# B&R Automation Studio project VisionSample (part 8)

#### ViSaveImgOnPlc.st
```iecst
// Note: This FBK needs to be called at least once in the INIT of the task to alloc memory (restriction of AsMem)
FUNCTION_BLOCK ViSaveImgOnPlc
	IF MemInfo.SvgAdr = 0 THEN // This will only be done once in the INIT of the task
		// Create memory for uploading and transforming image
		// Size: a 5MP picture in bmp format has less than 6.000.000 Bytes. A SVG with bas64 conversion maximum the 4/3 size.
		MemInfo.UploadSize			:= 6000000;		// Upload of the picture data with httpClient
		MemInfo.SvgHeaderSize		:= 2000; 		// Fileheader, ...
		MemInfo.CrosshSize			:= 18000; 		// Crosshairs, Texts, ...
		MemInfo.SvgSize				:= MemInfo.UploadSize * 4 / 3 + MemInfo.SvgHeaderSize + MemInfo.CrosshSize;
		AsMemPartCreate_0.enable	:= TRUE;
		AsMemPartCreate_0.len		:= MemInfo.UploadSize + MemInfo.SvgSize + MemInfo.CrosshSize + 1000; // 1000 Bytes for AsMemPart stuff/header
		AsMemPartCreate_0();
		IF AsMemPartCreate_0.status = ERR_OK THEN
			// Upload mem for loading the image from camera to plc
			AsMemPartAllocClear_0.len		:= MemInfo.UploadSize;
			AsMemPartAllocClear_0(enable := TRUE, ident := AsMemPartCreate_0.ident);
			IF AsMemPartAllocClear_0.status = ERR_OK THEN
				MemInfo.UploadAdr			:= AsMemPartAllocClear_0.mem;
			END_IF
			// Svg mem for creating the svg file including the image
			AsMemPartAllocClear_0.len		:= MemInfo.SvgSize;
			AsMemPartAllocClear_0(enable := TRUE, ident := AsMemPartCreate_0.ident);
			IF AsMemPartAllocClear_0.status = ERR_OK THEN
				MemInfo.SvgAdr 				:= AsMemPartAllocClear_0.mem;
			END_IF
			// Mem for creating the crosshaurs
			AsMemPartAllocClear_0.len		:= MemInfo.CrosshSize;
			AsMemPartAllocClear_0(enable := TRUE, ident := AsMemPartCreate_0.ident);
			IF AsMemPartAllocClear_0.status = ERR_OK THEN
				MemInfo.CrosshAdr			:= AsMemPartAllocClear_0.mem;
			END_IF
		END_IF
	END_IF
	IF NOT Enable THEN
		Status := ERR_FUB_ENABLE_FALSE;
		Step := 0;
		RETURN;
	END_IF
	CASE Step OF
		0:
			Status := ERR_FUB_BUSY;
			IF MemInfo.UploadAdr <> 0 AND MemInfo.SvgAdr <> 0 AND MemInfo.CrosshAdr <> 0 THEN
				Step := 1;
			END_IF
		1: // Initialization
			ACTION_InitTexts;
			brsmemcpy(ADR(b64key), ADR('ABCDEFGHIJKLMNOPQRSTUVWXYZabcdefghijklmnopqrstuvwxyz0123456789+/'), SIZEOF(b64key));
			// Generate new filenames
			DTGetTime_0(enable := TRUE);
			DT_TO_DTStructure(DTGetTime_0.DT1, ADR(DTStructure_0));
			FileNameImg := CFG.DirName;
			brsstrcat(ADR(FileNameImg), ADR('/'));
			tmpStr1 := UINT_TO_STRING(DTStructure_0.year);
			brsstrcat(ADR(FileNameImg), ADR(tmpStr1));
			brsstrcat(ADR(FileNameImg), ADR('_'));
			tmpStr1 := USINT_TO_STRING(DTStructure_0.month);
			IF(DTStructure_0.month < 10) THEN
				brsstrcat(ADR(FileNameImg), ADR('0'));
			END_IF
			brsstrcat(ADR(FileNameImg), ADR(tmpStr1));
			brsstrcat(ADR(FileNameImg), ADR('_'));
			tmpStr1 := USINT_TO_STRING(DTStructure_0.day);
			IF(DTStructure_0.day < 10) THEN
				brsstrcat(ADR(FileNameImg), ADR('0'));
			END_IF
			brsstrcat(ADR(FileNameImg), ADR(tmpStr1));
			brsstrcat(ADR(FileNameImg), ADR('_'));
			tmpStr1 := USINT_TO_STRING(DTStructure_0.hour);
			IF(DTStructure_0.hour < 10) THEN
				brsstrcat(ADR(FileNameImg), ADR('0'));
			END_IF
			brsstrcat(ADR(FileNameImg), ADR(tmpStr1));
			brsstrcat(ADR(FileNameImg), ADR('_'));
			tmpStr1 := USINT_TO_STRING(DTStructure_0.minute);
			IF(DTStructure_0.minute < 10) THEN
				brsstrcat(ADR(FileNameImg), ADR('0'));
			END_IF
			brsstrcat(ADR(FileNameImg), ADR(tmpStr1));
			brsstrcat(ADR(FileNameImg), ADR('_'));
			tmpStr1 := USINT_TO_STRING(DTStructure_0.second);
			IF(DTStructure_0.second < 10) THEN
				brsstrcat(ADR(FileNameImg), ADR('0'));
			END_IF
			brsstrcat(ADR(FileNameImg), ADR(tmpStr1));
			brsstrcat(ADR(FileNameImg), ADR('.'));
			brsstrcpy(ADR(FileNameSvg), ADR(FileNameImg)); // Same filename but differend ending
			IF CFG.Format = 0 THEN
				brsstrcat(ADR(FileNameImg), ADR('jpg'));
			ELSE
				brsstrcat(ADR(FileNameImg), ADR('bmp'));
			END_IF
			brsstrcat(ADR(FileNameSvg), ADR('svg'));
			// Create URI and Host
			URI := '/';
			IF CFG.Format = 0 THEN
				brsstrcat(ADR(URI), ADR('jpg'));
				brsstrcat(ADR(URI), ADR('?q='));
				brsitoa(CFG.QualityJPG, ADR(tmpStr1));
				brsstrcat(ADR(URI), ADR(tmpStr1));
			ELSE
				brsstrcat(ADR(URI), ADR('bmp'));
			END_IF
			Host := CFG.PlkIPWithoutNode;
			brsitoa(PowerlinkNode, ADR(tmpStr1));
			brsstrcat(ADR(Host), ADR(tmpStr1));
			DiagStartTime := clock_ms();
			Step := 10;

		10: // Reset timer and HTTP client
			TON_ReloadTimeout(IN := FALSE);
			httpClient_0(enable := FALSE, abort := FALSE, send := FALSE);
			IF httpClient_0.status = ERR_FUB_ENABLE_FALSE THEN
				Step := 11;
			END_IF

		11: // Wait for response
			TON_ReloadTimeout(IN := TRUE, PT := T#10s); // Time out when no response after 10s
			RequestHeader.keepAlive			:= 'timeout=5, max=100';
			httpClient_0.enable				:= TRUE;
			httpClient_0.send				:= TRUE;
			httpClient_0.method 			:= httpMETHOD_GET;
			httpClient_0.option 			:= httpOPTION_HTTP_11;
			httpClient_0.hostPort			:= 8080;
			httpClient_0.pHost 				:= ADR(Host);
			httpClient_0.pUri 				:= ADR(URI);
			httpClient_0.pResponseData 		:= MemInfo.UploadAdr;
			httpClient_0.responseDataSize	:= MemInfo.UploadSize;
			httpClient_0.pRequestHeader		:= ADR(RequestHeader);
			httpClient_0();
			IF httpClient_0.status = ERR_OK AND httpClient_0.responseDataLen <> 0 THEN
				UploadedImgSize				:= httpClient_0.responseDataLen;
				httpClient_0(send := FALSE);
				IF UploadedImgSize < 100 THEN // No image available. Hint: In case of no image there will be sent 86 Bytes with an html error text
					Status := ERR_NO_IMAGE;
					Step := 0;
				ELSE
					IF CFG.UploadBmpJpg THEN
						Step := 20; // save the image (bmp or jpg)
					ELSE
						Step := 30; // directly upload the svg
					END_IF
				END_IF
			ELSIF httpClient_0.status <> ERR_FUB_BUSY AND httpClient_0.status <> 0 THEN
				httpClientErrorStatus := httpClient_0.status;
				Step := 19;
			ELSIF TON_ReloadTimeout.Q THEN // Timout! httpClient takes too long, so abort
				Status := ERR_NO_IMAGE;
				Step := 0;
			END_IF
		19: // httpclient Error
			httpClient_0.enable	:= TRUE;
			httpClient_0.send	:= FALSE;
			httpClient_0.abort	:= TRUE;
			httpClient_0();
			IF httpClient_0.status <> ERR_FUB_BUSY THEN
				httpClient_0.abort := FALSE;
				httpClient_0();
				Status := httpClientErrorStatus;
				Step := 0;
			END_IF

		20: // Save bmp/jpg file
			DiagTime.BeginSaveBMPJPG := clock_ms() - DiagStartTime;
			FileCreate_0.enable		:= TRUE;
			FileCreate_0.pDevice	:= ADR(CFG.FileDevice);
			FileCreate_0.pFile		:= ADR(FileNameImg);
			FileCreate_0();
			IF FileCreate_0.status = ERR_OK THEN
				Step := 21;
			ELSIF FileCreate_0.status <> ERR_FUB_BUSY THEN
				Status := FileCreate_0.status;
				Step := 0;
			END_IF
		21:
			FileWrite_0.enable		:= TRUE;
			FileWrite_0.ident		:= FileCreate_0.ident;
			FileWrite_0.offset		:= 0;
			FileWrite_0.pSrc		:= MemInfo.UploadAdr;
			FileWrite_0.len			:= UploadedImgSize;
			FileWrite_0();
			IF FileWrite_0.status = ERR_OK THEN
				Step := 22;
			ELSIF FileWrite_0.status <> ERR_FUB_BUSY THEN
				Status := FileWrite_0.status;
				Step := 0;
			END_IF
		22:
			FileClose_0.enable		:= TRUE;
			FileClose_0.ident		:= FileCreate_0.ident;
			FileClose_0();
			IF FileClose_0.status = ERR_OK THEN
				DiagTime.EndSaveBMPJPG := clock_ms() - DiagStartTime;
				IF CFG.UploadSVG THEN
					Step := 30;
				ELSE // ready
					Status := 0;
					Step := 0;
				END_IF
			ELSIF FileClose_0.status <> ERR_FUB_BUSY THEN
				Status := FileClose_0.status;
				Step := 0;
			END_IF

		30: // Create SVG file with image and crosshair/texts
			DiagTime.BeginSVG := clock_ms() - DiagStartTime;
			b64neededOutput	:= (UploadedImgSize/3)*4 + BOOL_TO_UDINT(UDINT_TO_BOOL(UploadedImgSize MOD 3))*4;
			IF b64neededOutput < MemInfo.SvgSize - MemInfo.SvgHeaderSize - MemInfo.CrosshSize THEN
				brsmemset(MemInfo.SvgAdr, 0, MemInfo.SvgSize); // clear complete memory
				// Prepare the svg header up to the base64 picture data
				brsstrcpy(MemInfo.SvgAdr, ADR(SvgTexts.ContentStart));
				brsstrcat(MemInfo.SvgAdr, ADR(FileNameSvg));
				brsstrcat(MemInfo.SvgAdr, ADR(SvgTexts.ContentAfterTitle));
				IF CFG.Format = 0 THEN
					brsstrcat(MemInfo.SvgAdr, ADR('jpg'));
				ELSE
					brsstrcat(MemInfo.SvgAdr, ADR('bmp'));
				END_IF
				brsstrcat(MemInfo.SvgAdr, ADR(SvgTexts.ContentBase64));
				Step := 31;
			ELSE
				Status := ERR_BUFF_SVG;
				Step := 0;
			END_IF

		31: // Code picture data with Base64 to embedd the picture into a svg file
			b64AdrInBuffer	:= MemInfo.UploadAdr; // Original bmp or jpg picture
			b64AdrOutBuffer	:= MemInfo.SvgAdr + brsstrlen(MemInfo.SvgAdr); // Write to the end of the actual svg data
			b64actposIN		:= b64AdrInBuffer;
			b64actposOUT	:= b64AdrOutBuffer;
			Step := 32;
		32: // Convert
			FOR i := 0 TO CFG.ConvertCycles DO
				IF b64actposIN < b64AdrInBuffer + UploadedImgSize THEN
					b64blockLen := UDINT_TO_USINT(LIMIT(0, b64AdrInBuffer + UploadedImgSize - b64actposIN, 3));
					b64in ACCESS b64actposIN;
					b64out ACCESS b64actposOUT;
					b64out[0]		:= b64key[ SHR(b64in[0],2) ];	// always
					IF b64blockLen = 1 THEN
						b64out[1]	:= b64key[ SHL((b64in[0] AND 16#03),4)];
						b64out[2]	:= 61;	// 61 = '='
						b64out[3]	:= 61;	// 61 = '='
					ELSIF b64blockLen = 2 THEN
						b64out[1]	:= b64key[ SHL((b64in[0] AND 16#03),4) OR SHR(b64in[1],4) ];
						b64out[2]	:= b64key[ SHL((b64in[1] AND 16#0F),2)];
						b64out[3]	:= 61;	// 61 = '='
					ELSIF b64blockLen = 3 THEN
						b64out[1]	:= b64key[ SHL((b64in[0] AND 16#03),4) OR SHR(b64in[1],4) ];
						b64out[2]	:= b64key[ SHL((b64in[1] AND 16#0F),2) OR SHR(b64in[2],6) ];
						b64out[3]	:= b64key[ b64in[2] AND 16#3F ];
					END_IF
					b64actposIN		:= b64actposIN + 3;
					b64actposOUT	:= b64actposOUT + 4;
				ELSE
					Step := 33;
					EXIT;
				END_IF
			END_FOR

		33: // Prepare the second part after base64 picture data
			brsmemset(MemInfo.CrosshAdr, 0, MemInfo.CrosshSize);
			brsstrcat(MemInfo.CrosshAdr, ADR(SvgTexts.ContentBeginJS));
			brsstrcat(MemInfo.CrosshAdr, ADR(CrossHairInfo[1].DataVis));
			brsstrcat(MemInfo.CrosshAdr, ADR(SvgTexts.ContentBetween1));
			FirstElement := TRUE;
			FOR i := 1 TO MAX_NUM_RESULTS DO
				IF CrossHairInfo[i].CrosshairTopLeftX <> 0 AND CrossHairInfo[i].CrosshairTopLeftY <> 0 THEN
					IF FirstElement THEN
						FirstElement := FALSE;
					ELSE
						brsstrcat(MemInfo.CrosshAdr, ADR(SvgTexts.ContentBetween2)); // Needed between the elements
					END_IF
					brsstrcat(MemInfo.CrosshAdr, ADR(CrossHairInfo[i].Data));
				END_IF
			END_FOR
			brsstrcat(MemInfo.CrosshAdr, ADR(SvgTexts.ContentEndJS));

			// Create the crosshairs
			FOR i := 1 TO MAX_NUM_RESULTS DO
				IF CrossHairInfo[i].CrosshairTopLeftX <> 0 AND CrossHairInfo[i].CrosshairTopLeftY <> 0 THEN
					brsstrcat(MemInfo.CrosshAdr, ADR(SvgTexts.ContentCrossHairBegin));
					brsitoa(i, ADR(tmpStr1));
					brsstrcat(MemInfo.CrosshAdr, ADR(tmpStr1));
					brsstrcat(MemInfo.CrosshAdr, ADR(SvgTexts.ContentCrossHairMiddle));
					brsitoa(REAL_TO_DINT(CrossHairInfo[i].CrosshairTopLeftX), ADR(tmpStr1));
					brsstrcat(MemInfo.CrosshAdr, ADR(tmpStr1));
					brsstrcat(MemInfo.CrosshAdr, ADR(','));
					brsitoa(REAL_TO_DINT(CrossHairInfo[i].CrosshairTopLeftY), ADR(tmpStr1));
					brsstrcat(MemInfo.CrosshAdr, ADR(tmpStr1));
					brsstrcat(MemInfo.CrosshAdr, ADR(') rotate('));
					brsitoa(REAL_TO_DINT(CrossHairInfo[i].CrosshairRotateCenter), ADR(tmpStr1));
					brsstrcat(MemInfo.CrosshAdr, ADR(tmpStr1));
					brsstrcat(MemInfo.CrosshAdr, ADR(','));
					brsitoa(REAL_TO_DINT(CrossHairInfo[i].CrosshairSizeScaled / 2), ADR(tmpStr1));
					brsstrcat(MemInfo.CrosshAdr, ADR(tmpStr1));
					brsstrcat(MemInfo.CrosshAdr, ADR(','));
					brsstrcat(MemInfo.CrosshAdr, ADR(tmpStr1));
					brsstrcat(MemInfo.CrosshAdr, ADR(') scale('));
					brsitoa(REAL_TO_DINT(CrossHairInfo[i].CrosshairScale), ADR(tmpStr1));
					brsstrcat(MemInfo.CrosshAdr, ADR(tmpStr1));
					brsstrcat(MemInfo.CrosshAdr, ADR(','));
					brsstrcat(MemInfo.CrosshAdr, ADR(tmpStr1));
					brsstrcat(MemInfo.CrosshAdr, ADR(SvgTexts.ContentCrossHairEnd));
				END_IF
			END_FOR
			brsstrcat(MemInfo.CrosshAdr, ADR(SvgTexts.ContentCrossHairRed));
			// Create the indices
			FOR i := 1 TO MAX_NUM_RESULTS DO
				IF CrossHairInfo[i].CrosshairTopLeftX <> 0 AND CrossHairInfo[i].CrosshairTopLeftY <> 0 THEN
					brsstrcat(MemInfo.CrosshAdr, ADR(SvgTexts.ContentCrossHairIndex));
				END_IF
			END_FOR
			brsstrcat(MemInfo.CrosshAdr, ADR(SvgTexts.ContentEnd));
			Step := 41;
		41:
			brsstrcat(MemInfo.SvgAdr, MemInfo.CrosshAdr);
			Step := 50;
		50:
			DiagTime.BeginSVGSave := clock_ms() - DiagStartTime;
			FileCreate_0.enable		:= TRUE;
			FileCreate_0.pDevice	:= ADR(CFG.FileDevice);
			FileCreate_0.pFile		:= ADR(FileNameSvg);
			FileCreate_0();
			IF FileCreate_0.status = ERR_OK THEN
				Step := 51;
			ELSIF FileCreate_0.status <> ERR_FUB_BUSY THEN
				Status := FileCreate_0.status;
				Step := 0;
			END_IF
		51:
			FileWrite_0.enable		:= TRUE;
			FileWrite_0.ident		:= FileCreate_0.ident;
			FileWrite_0.offset		:= 0;
			FileWrite_0.pSrc		:= MemInfo.SvgAdr;
			FileWrite_0.len			:= brsstrlen(MemInfo.SvgAdr);
			FileWrite_0();
			IF FileWrite_0.status = ERR_OK THEN
				Step := 52;
			ELSIF FileWrite_0.status <> ERR_FUB_BUSY THEN
				Status := FileWrite_0.status;
				Step := 0;
			END_IF
		52:
			FileClose_0.enable		:= TRUE;
			FileClose_0.ident		:= FileCreate_0.ident;
			FileClose_0();
			IF FileClose_0.status = ERR_OK THEN
				DiagTime.EndSVGSave := clock_ms() - DiagStartTime;
				Status := 0;
				Step := 0;
			ELSIF FileClose_0.status <> ERR_FUB_BUSY THEN
				Status := FileClose_0.status;
				Step := 0;
			END_IF
	END_CASE
END_FUNCTION_BLOCK
```

#### ViShowImgOnVC4.st
```iecst
// Note: This FBK needs to be called at least once in the INIT of the task to alloc memory (restriction of AsMem)
FUNCTION_BLOCK ViShowImgOnVC4
	IF MemInfo.UploadBmp8Adr = 0 THEN // This will only be done once in the INIT of the task
		// Create memory for uploading and transforming image
		// Size: a 5MP picture in bmp format has less than 6.000.000 Bytes. A SVG with bas64 conversion maximum the 4/3 size.
		MemInfo.UploadBmp8Size		:= 6000000;		// Upload of the picture data with httpClient
		MemInfo.Bmp24Size			:= 18000000; 	// The 24bit img could be 3 times bigger
		AsMemPartCreate_0.enable	:= TRUE;
		AsMemPartCreate_0.len		:= MemInfo.UploadBmp8Size + MemInfo.Bmp24Size + 1000; // 1000 Bytes for AsMemPart stuff/header
		AsMemPartCreate_0();
		IF AsMemPartCreate_0.status = ERR_OK THEN
			// Upload mem for loading the image from camera to plc
			AsMemPartAllocClear_0.len		:= MemInfo.UploadBmp8Size;
			AsMemPartAllocClear_0(enable := TRUE, ident := AsMemPartCreate_0.ident);
			IF AsMemPartAllocClear_0.status = ERR_OK THEN
				MemInfo.UploadBmp8Adr		:= AsMemPartAllocClear_0.mem;
			END_IF
			// Bmp24 mem for creating the new image
			AsMemPartAllocClear_0.len		:= MemInfo.Bmp24Size;
			AsMemPartAllocClear_0(enable := TRUE, ident := AsMemPartCreate_0.ident);
			IF AsMemPartAllocClear_0.status = ERR_OK THEN
				MemInfo.Bmp24Adr 			:= AsMemPartAllocClear_0.mem;
			END_IF
		END_IF
	END_IF
	IF NOT Enable THEN
		HTMLStreamContent	:= '<p>Ready</p>';
		RefreshDone			:= FALSE;
		Status := ERR_FUB_ENABLE_FALSE;
		Step := 0;
		RETURN;
	END_IF
	CASE Step OF
		0:
			RefreshDone := FALSE;
			Status := ERR_FUB_BUSY;
			IF MemInfo.UploadBmp8Adr <> 0 AND MemInfo.Bmp24Adr <> 0 THEN
				IF RefreshImage THEN
					Step := 1;
				END_IF
			END_IF
		1: // Initialization
			CreateVC4HTML;
			FileNameBmp24Bit	:= 'http://localhost/CamImgVC4.bmp';
			FileNameBmp24BitDir	:= 'web/CamImgVC4.bmp';
			// Create URI and Host
			URI := '/bmp';
			Host := CFG.PlkIPWithoutNode;
			brsitoa(PowerlinkNode, ADR(tmpStr1));
			brsstrcat(ADR(Host), ADR(tmpStr1));
			HTMLStreamContent := '<p>Please wait... image will be loaded...</p>';
			Step := 10;
		10: // Reset timer and HTTP client
			TON_Timeout(IN := FALSE);
			httpClient_0(enable := FALSE, abort := FALSE, send := FALSE);
			IF httpClient_0.status = ERR_FUB_ENABLE_FALSE THEN
				Step := 11;
			END_IF

		11: // Wait for response
			TON_Timeout(IN := TRUE, PT := T#10s); // Time out when no response after 10s
			RequestHeader.keepAlive			:= 'timeout=5, max=100';
			httpClient_0.enable				:= TRUE;
			httpClient_0.send				:= TRUE;
			httpClient_0.method 			:= httpMETHOD_GET;
			httpClient_0.option 			:= httpOPTION_HTTP_11;
			httpClient_0.hostPort			:= 8080;
			httpClient_0.pHost 				:= ADR(Host);
			httpClient_0.pUri 				:= ADR(URI);
			httpClient_0.pResponseData 		:= MemInfo.UploadBmp8Adr;
			httpClient_0.responseDataSize	:= MemInfo.UploadBmp8Size;
			httpClient_0.pRequestHeader		:= ADR(RequestHeader);
			httpClient_0();
			IF httpClient_0.status = ERR_OK AND httpClient_0.responseDataLen <> 0 THEN
				FileSizeIn8Bit				:= httpClient_0.responseDataLen;
				httpClient_0(send := FALSE);
				IF FileSizeIn8Bit < 100 THEN // No image available. Hint: In case of no image there will be sent 86 Bytes with an html error text
					HTMLStreamContent := '<p>No image found on the camera</p>';
					Status := ERR_NO_IMAGE;
					Step := 50;
				ELSE
					Step := 20;
				END_IF
			ELSIF httpClient_0.status <> ERR_FUB_BUSY AND httpClient_0.status <> 0 THEN
				httpClientErrorStatus := httpClient_0.status;
				Step := 19;
			ELSIF TON_Timeout.Q THEN // Timout! httpClient takes too long, so abort
				HTMLStreamContent := '<p>Timeout while loading image</p>';
				Status := ERR_NO_IMAGE;
				Step := 50;
			END_IF
		19: // httpclient Error
			httpClient_0.enable	:= TRUE;
			httpClient_0.send	:= FALSE;
			httpClient_0.abort	:= TRUE;
			httpClient_0();
			IF httpClient_0.status <> ERR_FUB_BUSY THEN
				httpClient_0.abort := FALSE;
				httpClient_0();
				Status := httpClientErrorStatus;
				Step := 50;
			END_IF

		20: // Convert image from 8 bit bmp with color table to 24 bit bmp image
			brsmemcpy(ADR(Bmp8Bit)+2, MemInfo.UploadBmp8Adr, SIZEOF(Bmp8Bit)); // Use the read data
			brsmemcpy(ADR(Bmp24Bit), ADR(Bmp8Bit), SIZEOF(Bmp24Bit)); // Copy the header, but not the colour data
			// Change and add fileheader
			Bmp24Bit.InfoHeader.biBitCount	:= 24;
			Bmp24Bit.FileHeader.bfOffBits	:= SIZEOF(Bmp24Bit)-2;
			brsmemcpy(MemInfo.Bmp24Adr, ADR(Bmp24Bit)+2, SIZEOF(Bmp24Bit)-2);
			// Generate pixels
			BytesPerLine := Bmp24Bit.InfoHeader.biWidth;
			IF BytesPerLine MOD 4 > 0 THEN // Add fill bytes if necessary. The lengt of a line is always a multiple of 4.
				BytesPerLine := BytesPerLine + (4 - BytesPerLine MOD 4);
			END_IF
			IF Bmp8Bit.FileHeader.bfOffBits > (14+40+4*255) AND BytesPerLine > 0 AND ABS(Bmp24Bit.InfoHeader.biHeight) > 0 THEN // Header 14+40 + ColorTable
				PixelSourceAdr	:= MemInfo.UploadBmp8Adr + Bmp8Bit.FileHeader.bfOffBits;
				PixelDestAdr	:= MemInfo.Bmp24Adr + SIZEOF(Bmp24Bit)-2; // directly start after the header. -2 because of two fillbyts at the beginning
				BytesRemaining	:= BytesPerLine * ABS(Bmp24Bit.InfoHeader.biHeight);
				Step := 21;
			ELSE
				Status := ERR_DATA_BMP;
				Step := 50;
			END_IF
		21:
			FOR i := 0 TO CFG.ConvertCycles DO
				PixelSourceColor ACCESS PixelSourceAdr;
				PixelDestColor ACCESS PixelDestAdr;
				PixelDestColor.Blue		:= Bmp8Bit.ColorTable[PixelSourceColor].Blue;
				PixelDestColor.Green	:= Bmp8Bit.ColorTable[PixelSourceColor].Green;
				PixelDestColor.Red		:= Bmp8Bit.ColorTable[PixelSourceColor].Red;
				BytesRemaining := BytesRemaining - 1;
				IF BytesRemaining = 0 THEN
					Step := 30;
					EXIT;
				ELSE
					PixelSourceAdr		:= PixelSourceAdr + 1;
					PixelDestAdr		:= PixelDestAdr + 3;
					IF PixelSourceAdr > MemInfo.UploadBmp8Adr + MemInfo.UploadBmp8Size - 1 OR PixelDestAdr + 2 > MemInfo.Bmp24Adr + MemInfo.Bmp24Size -1 THEN
						Status := ERR_BUFF_BMP;
						Step := 50;
						EXIT;
					END_IF
				END_IF
			END_FOR

		30: // Save content to a bmp file
			FileDelete_0.enable		:= TRUE;
			FileDelete_0.pDevice	:= ADR(CFG.FileDevice);
			FileDelete_0.pName		:= ADR(FileNameBmp24BitDir);
			FileDelete_0();
			IF FileDelete_0.status = ERR_OK OR FileDelete_0.status = fiERR_FILE_NOT_FOUND THEN
				Step := 31;
			ELSIF FileDelete_0.status <> ERR_FUB_BUSY THEN
				Status := FileDelete_0.status;
				Step := 100;
			END_IF
		31:
			FileCreate_0.enable		:= TRUE;
			FileCreate_0.pDevice	:= ADR(CFG.FileDevice);
			FileCreate_0.pFile		:= ADR(FileNameBmp24BitDir);
			FileCreate_0();
			IF FileCreate_0.status = ERR_OK THEN
				Step := 32;
			ELSIF FileCreate_0.status <> ERR_FUB_BUSY THEN
				Status := FileCreate_0.status;
				Step := 100;
			END_IF
		32:
			FileWrite_0.enable		:= TRUE;
			FileWrite_0.ident		:= FileCreate_0.ident;
			FileWrite_0.pSrc		:= MemInfo.Bmp24Adr;
			FileWrite_0.len			:= MIN(MemInfo.Bmp24Size, PixelDestAdr - MemInfo.Bmp24Adr);
			FileWrite_0();
			IF FileWrite_0.status = ERR_OK THEN
				Step := 33;
			ELSIF FileWrite_0.status <> ERR_FUB_BUSY THEN
				Status := FileWrite_0.status;
				Step := 100;
			END_IF
		33:
			FileClose_0.enable	:= TRUE;
			FileClose_0.ident	:= FileCreate_0.ident;
			FileClose_0();
			IF FileClose_0.status = ERR_OK THEN
				Step := 40;
			ELSIF FileClose_0.status <> ERR_FUB_BUSY THEN
				Status := FileClose_0.status;
				Step := 100;
			END_IF

		40: // Create content for VC4 html control element
			ImgHeight_px := UDINT_TO_UINT(UINT_TO_UDINT(ImgWidthInVC4_px) *1024 / 1280);
			brsstrcpy(ADR(HTMLStreamContent), ADR(VC4HTML[0]));
			brsitoa(ImgWidthInVC4_px, ADR(tmpStr1));
			brsstrcat(ADR(HTMLStreamContent), ADR(tmpStr1));
			brsstrcat(ADR(HTMLStreamContent), ADR(VC4HTML[1]));
			brsitoa(ImgHeight_px, ADR(tmpStr1));
			brsstrcat(ADR(HTMLStreamContent), ADR(tmpStr1));
			brsstrcat(ADR(HTMLStreamContent), ADR(VC4HTML[2]));
			brsstrcat(ADR(HTMLStreamContent), ADR(FileNameBmp24Bit));
			brsstrcat(ADR(HTMLStreamContent), ADR(VC4HTML[3]));
			Status := 0;
			Step := 50;

		50:
			RefreshDone := TRUE;
			IF NOT RefreshImage THEN
				RefreshDone := FALSE;
				Step := 0;
			END_IF
	END_CASE
END_FUNCTION_BLOCK
```

#### CrosshairDetails.st
```iecst
FUNCTION CrosshairDetailsValue
	IF NOT TextAlignment THEN // left
		tmpStr:= '<tspan text-anchor="start" class="text" x="10" dy="32">';
	ELSE // right
		tmpStr:= '<tspan text-anchor="end" class="text" x="1270" dy="32">';
	END_IF
	brsstrcat(strTarget, ADR(tmpStr));
	brsstrcat(strTarget, strText);
	brsftoa(fValue, ADR(tmpStr));
	brsstrcat(strTarget, ADR(tmpStr));
	brsstrcat(strTarget, ADR('</tspan> '));
	CrosshairDetailsValue := TRUE;
END_FUNCTION
FUNCTION CrosshairDetailsText
	IF NOT TextAlignment THEN // left
		tmpStr:= '<tspan text-anchor="start" class="text" x="10" dy="32">';
	ELSE // right
		tmpStr:= '<tspan text-anchor="end" class="text" x="1270" dy="32">';
	END_IF
	brsstrcat(strTarget, ADR(tmpStr));
	brsstrcat(strTarget, strText);
	brsstrcat(strTarget, adrText);
	brsstrcat(strTarget, ADR('</tspan> '));
	CrosshairDetailsText := TRUE;
END_FUNCTION
```

### Program Logical/old/Vi_image

#### Types.typ
```iecst
TYPE
	VIStep_Enum :
		(
		VISTEP_WAIT,
		VISTEP_CREATE_DIR,
		VISTEP_DELETE_DIR,
		VISTEP_DELETE_IMAGE,
		VISTEP_REFRESH_IMG_LIST,
		VISTEP_DOWNLOAD_IMAGE,
		VISTEP_SAVE_IMG_ON_PLC,
		VISTEP_ERR
		);
	SvgTexts_Type : 	STRUCT
		ContentStart : STRING[500];
		ContentAfterTitle : STRING[200];
		ContentBase64 : STRING[200];
		ContentBeginJS : STRING[2000];
		ContentBetween1 : STRING[200];
		ContentBetween2 : STRING[200];
		ContentEndJS : STRING[3000];
		ContentCrossHairBegin : STRING[200];
		ContentCrossHairMiddle : STRING[200];
		ContentCrossHairEnd : STRING[200];
		ContentCrossHairRed : STRING[200];
		ContentCrossHairIndex : STRING[200];
		ContentEnd : STRING[2000];
	END_STRUCT;
	DiagTime_Type : 	STRUCT
		Refresh : TIME;
		BeginSaveBMPJPG : TIME;
		EndSaveBMPJPG : TIME;
		BeginSVG : TIME;
		BeginSVGSave : TIME;
		EndSVGSave : TIME;
	END_STRUCT;
	MemInfoSave_Type : 	STRUCT
		UploadAdr : UDINT;
		UploadSize : UDINT; (*Upload of the picture data with httpClient*)
		SvgAdr : UDINT;
		SvgSize : UDINT;
		CrosshAdr : UDINT;
		CrosshSize : UDINT; (*Crosshairs, Texts, ...*)
		SvgHeaderSize : UDINT; (*Fileheader, ...*)
	END_STRUCT;
	MemInfoVC4_Type : 	STRUCT
		UploadBmp8Adr : UDINT;
		UploadBmp8Size : UDINT; (*Upload of the picture data with httpClient*)
		Bmp24Adr : UDINT;
		Bmp24Size : UDINT;
	END_STRUCT;
	typCrossHair : 	STRUCT  (*Cross hair data structure*)
		SvgTransformation : ARRAY[1..MAX_NUM_RESULTS]OF STRING[200] := [10('')]; (*Transformation string for paper widget*)
		SvgContent : ARRAY[1..MAX_NUM_RESULTS]OF STRING[1000]; (*Transformation string for paper widget*)
		SvgVisible : ARRAY[1..MAX_NUM_RESULTS]OF BOOL := [10(FALSE)];
		CFG : typCrossHairCfg;
		DetailsNo : USINT := 1;
		ShowCrosshair : BOOL := TRUE; (*Enable/Disable cross hairs*)
	END_STRUCT;
	typCrossHairCfg : 	STRUCT
		Scale : REAL := 1; (*Scale size of the cross hair*)
		PixelRatio : REAL := 100; (*Position value for one pixel*)
		Size : USINT := 80; (*Size of the cross hair in pixel*)
		Font : USINT := 35;
		RefSizeX : UINT := 1280; (*Size of the Webviewer Widget*)
		RefSizeY : UINT := 1024; (*Size of the Webviewer Widget*)
	END_STRUCT;
	typCrossHairInfo : 	STRUCT
		CrosshairTopLeftX : REAL; (*top left position of the crosshair in pixels*)
		CrosshairTopLeftY : REAL; (*top left position of the crosshair in pixels*)
		CrosshairRotateCenter : REAL; (*crosshair rotation around center in degrees*)
		CrosshairSizeScaled : REAL; (*crosshair size in pixel (in both directions)*)
		CrosshairScale : REAL;
		DataVis : STRING[80];
		Data : STRING[400];
		Text : STRING[1000];
	END_STRUCT;
	Bmp24Bit_Type : 	STRUCT
		FileHeader : BmpFileHeader_Type;
		InfoHeader : BmpInfoHeader_Type;
	END_STRUCT;
	Bmp8Bit_Type : 	STRUCT
		FileHeader : BmpFileHeader_Type;
		InfoHeader : BmpInfoHeader_Type;
		ColorTable : ARRAY[0..255]OF BmpColorTable_Type;
	END_STRUCT;
	BmpFileHeader_Type : 	STRUCT
		Fill : ARRAY[0..1]OF USINT;
		bfType : ARRAY[0..1]OF USINT;
		bfSize : UDINT;
		bfReserved : UDINT;
		bfOffBits : UDINT;
	END_STRUCT;
	BmpInfoHeader_Type : 	STRUCT
		biSize : UDINT;
		biWidth : DINT;
		biHeight : DINT;
		biPlanes : UINT;
		biBitCount : UINT;
		biCompression : UDINT;
		biSizeImage : UDINT;
		biXPelsPerMeter : DINT;
		biYPelsPerMeter : DINT;
		biClrUSer : UDINT;
		biClrImportant : UDINT;
	END_STRUCT;
	BmpColorTable_Type : 	STRUCT
		Blue : USINT;
		Green : USINT;
		Red : USINT;
		Fill : USINT;
	END_STRUCT;
	PixelDestColor_Type : 	STRUCT
		Blue : USINT;
		Green : USINT;
		Red : USINT;
	END_STRUCT;
END_TYPE
```

#### Actions.st
```iecst
ACTION ACTION_InitTexts:
SvgTexts.ContentStart :=
'<?xml version="1.0" encoding="UTF-8"?>
<!DOCTYPE svg PUBLIC "-//W3C//DTD SVG 1.1//EN" "http://www.w3.org/Graphics/SVG/1.1/DTD/svg11.dtd">
<svg xmlns="http://www.w3.org/2000/svg" xml:space="preserve" width="1280px" height="1024px" shape-rendering="geometricPrecision" text-rendering="geometricPrecision" image-rendering="optimizeQuality" fill-rule="nonzero" clip-rule="evenodd" viewBox="0 0 1280 1024" xmlns:xlink="http://www.w3.org/1999/xlink">
	<title>';
SvgTexts.ContentAfterTitle :=
'</title>
	<image
		xlink:href="data:image/';
SvgTexts.ContentBase64 :=
';base64,';
SvgTexts.ContentBeginJS :=
'"
		width="1280" height="1024"
		id="LoadedPicture"
		x="0" y="0"
	/>
	<defs>
		<style>
		  text {
		   pointer-events: none;
		   user-select: none;
		   -webkit-user-select: none;
		   -moz-user-select: none;
		  }
		</style>

		<symbol id="FadenkreuzBlau" fill="blue" stroke="blue" style="stroke-width:5">
			<use xlink:href="#Crosshair"/>
		</symbol>

		<symbol id="FadenkreuzRot" fill="red" stroke="red" style="stroke-width:5">
			<use xlink:href="#Crosshair"/>
		</symbol>

		<symbol id="Crosshair" >
			<path d="M 40,1 V 30 Z" id="up" />
			<path d="M 40,50 V 80 Z" id="down" />
			<path d="M 30,40 H 0 Z" id="left" />
			<path d="M 80,40 H 50 Z" id="right" />
			<circle style="fill:#000000; fill-opacity:0" cx="40" cy="40" r="25" />
		</symbol>

		<!-- Script -->
		<script type="text/javascript">
			<![CDATA[
			var blueCrosshairs, redCrosshair, indices, infoTxt;
			var amountElements;
			var actIndex = 1;
			var textInfo = ["Model ID: ", "Pos X: ", "Pos Y: ", "Orientation: ", "Clipped: ", "Gray: ", "Length: ", "Width: ", "Area: ", "Score: ", "Scale: ", "Grading: ", "Code Type: ", "Text: ", "Result: "];
			var visTextInfo = [';
SvgTexts.ContentBetween1 :=
'];
			var data = [
				[';
SvgTexts.ContentBetween2 :=
'],
				[';
SvgTexts.ContentEndJS :=
']
			];
			window.onload = function () {;
				blueCrosshairs 	= document.getElementsByName("crosshairBlue");
				redCrosshair	= document.getElementById("crosshairRed");
				indices			= document.getElementsByName("indice");
				infoTxt 		= document.getElementsByName("info");
				amountElements	= blueCrosshairs.length;
				let i;
				//fill and position indices
				for(i = 0; i < amountElements; i++) {
					indices[i].textContent = i + 1;
					let transformValues = blueCrosshairs[i].getAttribute("transform").match(/-?[\d.]+/g);
					indices[i].setAttribute("x", parseInt(transformValues[0]) + 85);
					indices[i].setAttribute("y", parseInt(transformValues[1]) + 35 );
				}
				//set visibility of information text
				for (i = 0; i< visTextInfo.length; i++ ){
					if (!visTextInfo[i]) {
						infoTxt[i].style.display = "none"
					}
				}
				//fill information text with first element and position red crosshair
				updateData(1);
				document.getElementById("crosshairRed").style.display = "inline";
				document.getElementById("infogroup").style.display = "inline";
			}

			function updateData(index) {
				index--; // Internal indices start at 0
				let i;
				for (i = 0; i< visTextInfo.length; i++ ){
					if (visTextInfo[i]) {
						infoTxt[i].textContent = textInfo[i] + data[index][i];
					}
				}
				document.getElementById("txtActElement").textContent = index + 1;
				//manipulate position of red crosshair
				let transform = blueCrosshairs[index].getAttribute("transform");
				redCrosshair.setAttribute("transform",transform);
				//set color of index number
				for(i = 0; i < amountElements; i++) {
					indices[i].setAttribute("fill","blue");
				}
				indices[index].setAttribute("fill","red");
			}
			function decreaseIndex(){
				actIndex--;
				if(actIndex < 1) actIndex = amountElements ;
				updateData(actIndex);
			}
			function increaseIndex(){
				actIndex++;
				if(actIndex > amountElements) actIndex = 1;
				updateData(actIndex);
			}
			]]>
		</script>
	</defs>

	<!-- blue crosshairs -->
';
SvgTexts.ContentCrossHairBegin :=
'	<use name="crosshairBlue" xlink:href="#FadenkreuzBlau" onclick="updateData(';
SvgTexts.ContentCrossHairMiddle :=
')" transform="translate(';
SvgTexts.ContentCrossHairEnd :=
')"/>
';
SvgTexts.ContentCrossHairRed :=
'
	<!-- red crosshair -->
	<use id="crosshairRed" xlink:href="#FadenkreuzRot" style="display: none"/>

	<!-- indices -->
';
SvgTexts.ContentCrossHairIndex :=
'	<text class="cText" font-size="22" font-family="Helvetica, Arial, sans-serif" > <tspan class="text" name="indice" fill="blue"></tspan></text>
';
SvgTexts.ContentEnd :=
'
	<g id="infogroup" transform="translate(20,30)" style="display: none">
		<!-- buttons -->
		<path d="M0,30, L60,60, L60,0, Z" stroke="black" fill="red" onclick="decreaseIndex()" style="stroke-width:5"/>
		<text id="txtActElement" fill="red" font-size="75" font-family="Helvetica, Arial, sans-serif" text-anchor="middle" x="102" y="55"></text>
		<path d="M150,60, L210,30, L150,0, Z" stroke="black" fill="red" onclick="increaseIndex()" style="stroke-width:5"/>

		<!-- informations -->
		<text class="cText" fill="red" font-size="35" font-family="Helvetica, Arial, sans-serif" x="0" y="80">
			<tspan class="text" name="info" x="0" dy="32"></tspan>
			<tspan class="text" name="info" x="0" dy="32"></tspan>
			<tspan class="text" name="info" x="0" dy="32"></tspan>
			<tspan class="text" name="info" x="0" dy="32"></tspan>
			<tspan class="text" name="info" x="0" dy="32"></tspan>
			<tspan class="text" name="info" x="0" dy="32"></tspan>
			<tspan class="text" name="info" x="0" dy="32"></tspan>
			<tspan class="text" name="info" x="0" dy="32"></tspan>
			<tspan class="text" name="info" x="0" dy="32"></tspan>
			<tspan class="text" name="info" x="0" dy="32"></tspan>
			<tspan class="text" name="info" x="0" dy="32"></tspan>
			<tspan class="text" name="info" x="0" dy="32"></tspan>
			<tspan class="text" name="info" x="0" dy="32"></tspan>
			<tspan class="text" name="info" x="0" dy="32"></tspan>
			<tspan class="text" name="info" x="0" dy="32"></tspan>
		</text>
	</g>
</svg>';
END_ACTION
ACTION ACTION_CreateHtmlFile:
HtmlFileContent1 :=
'<!DOCTYPE html>
<html lang="de">
	<head>
		<meta charset="utf-8" />
		<meta name="viewport" content="width=device-width, initial-scale=1.0" />
		<title>Camera Picture</title>
		<style>
			html, body{
				height: 100%;
				width: 100%;
				background: #C0C0C0;
				margin: 0;
				padding: 0;
			}
			img {
				width: 100%;
				height: auto;
				margin-left: auto;
				margin-right: auto;
			}
			div {
				height: 100%;
				width: 100%;
			}
		</style>
	</head>
	<body style="overflow: hidden">
		<div>
			<img id="imgError" src="VisionEye.png" />
			<img id="imgCamera" src="" />
			<script>
				function getParameterByName(param) {
					var url = window.location.href;
					var regex = new RegExp("[?&]" + param + "(=([^&#]*)|&|#|$$)"),
					results = regex.exec(url);
					if (!results) return null;
					if (!results[2]) return "";
					return decodeURIComponent(results[2].replace(/\+/g, " "));
				}
				var ImagePath 			= "http://';
HtmlFileContent2 :=
':8888/jpg";
				var ErrorImagePath 		= "VisionEye.png";
				var UpdateInterval_ms 	= 200;
				var MissingImgCtr		= 0;
				function updateImage() {
					document.getElementById("imgCamera").setAttribute("src", ImagePath + "?q=" + getParameterByName("q") + "&" + Math.random());
					var img = document.getElementById("imgCamera");
					var rot = getParameterByName("rot");
					var scale = getParameterByName("scale");
					if (scale == 0){
						scale = 1;
					}
					switch (rot) {
						case "0":
							move_x = 0;
							move_y = 0;
							break;
						case "90":
							move_x = img.height;
							move_y = 0;
							break;
						case "180":
							move_x = img.width;
							move_y = img.height;
							break;
						case "270":
							move_x = 0;
							move_y = img.width;
							break;
						default: //same as 0
							move_x = 0;
							move_y = 0;
					}
					document.getElementById("imgCamera").setAttribute("style", "transform-origin: 0% 0%; transform: scale(" + scale + ") translate(" + move_x + "px," + move_y + "px) rotate(" + rot + "deg);");
					if(img.naturalHeight !== 0 ) {
						MissingImgCtr = 0;
						showCameraImage() ;
					} else {
						MissingImgCtr++;
					}
					if(MissingImgCtr > 2){
						showErrorImage();
					}
					setTimeout(updateImage, UpdateInterval_ms);
				}
				showErrorImage();
				setTimeout(updateImage, UpdateInterval_ms);
				function showErrorImage() {
					var img = document.getElementById("imgError");
					img.style.display = "inline";
					var img = document.getElementById("imgCamera");
					img.style.display = "none";
				}
				function showCameraImage() {
					var img = document.getElementById("imgError");
					img.style.display = "none";
					var img = document.getElementById("imgCamera");
					img.style.display = "inline";
				}
			</script>
		</div>
	</body>
</html>';
END_ACTION
ACTION CreateVC4HTML:
VC4HTML[0] := '<!DOCTYPE html>
<html lang="de">
	<head>
		<meta charset="utf-8" />
		<meta name="viewport" content="width=device-width, initial-scale=1.0" />
		<title>Camera Picture</title>
	</head>
	<body >
		<img id="imgError" width="';
VC4HTML[1] := 'px" height="';
VC4HTML[2] := 'px" src="';
VC4HTML[3] := '" />
	</body>
</html>';
END_ACTION
```

#### Main.st
```iecst
// --------------------------------------------------------------------------------------------------------------------
// Vision image upload task
// - Stores the camera image on the file device media
// - Download of the image in the browser
// - Creates a html file to "resize" thei image for the mappview visualization (every size of the picuture matches the visu size)
// - Draw crosshairs
// Version 2.2
// --------------------------------------------------------------------------------------------------------------------
PROGRAM _INIT
	IF RemCfgImage.ConvertCycles = 0 THEN 								// Invalid --> use default values
		gVisionImage.CFG.FileDevice 		:= DEVICE_NAME;				// File device name where the images are stored
		gVisionImage.CFG.DirName			:= 'Vision';				// Directory used for images
		gVisionImage.CFG.PlkIPWithoutNode	:= '192.168.200.';			// IP adress of the plk interface, where the camera is connected to (see PLK settings), without the node (last part). Example: "192.168.200.0"
		gVisionImage.CFG.EthDevice			:= 'IF2';					// Device path of the PLCs ETH address
		gVisionImage.CFG.ConvertCycles		:= 10000;					// Conversioncycles per step (TK8 call). Use higer value on high performance CPU, use lower values on low performance CPU or in case of cycle time violations
		gVisionImage.CFG.Format				:= 0;						// Image type, use 0 for JPEG, 1 for bitmap
		gVisionImage.CFG.QualityJPG			:= 80;						// Quality for JPG images, larger numbers produce better images. Allowed values: 0 to 100, but values < ca 10 makes no sense
		gVisionImage.CFG.UploadBmpJpg		:= TRUE;
		gVisionImage.CFG.UploadSVG			:= TRUE;
		gVisionImage.CFG.ImageRotation_deg	:= 0;
		gVisionImage.CFG.MainPageQualityJPG	:= 30;
	ELSE
		brsmemcpy(ADR(gVisionImage.CFG), ADR(RemCfgImage), SIZEOF(RemCfgImage)); // Restore default values from remanent memory
	END_IF
	gVisionImage.CMD.CreateDir	:= TRUE;
	visSelectedImage			:= '';
	// Call FBKs which interanally alloc memory once in the INIT
	ViDownloadImage_0();
	ViSaveImgOnPlc_0();
	// Get IP address
	CfgGetIPAddr_0.enable		:= TRUE;
	CfgGetIPAddr_0.Len			:= SIZEOF(gVisionImage.CFG.EthIP);
	CfgGetIPAddr_0.pDevice		:= ADR(gVisionImage.CFG.EthDevice);
	CfgGetIPAddr_0.pIPAddr		:= ADR(gVisionImage.CFG.EthIP);
	CfgGetIPAddr_0();
	// Proxy server settings
	TcpForward_0.ServerPort := 8888;
	TcpForward_0.ConnectToPort := 8080 ;
END_PROGRAM
PROGRAM _CYCLIC
	CASE Step OF
		VISTEP_WAIT: // Wait for new upload command
			IF gVisionImage.CMD.CreateDir THEN // Create the image directory on user partition (if it does not exist)
				gVisionImage.DAT.Status := ERR_FUB_BUSY;
				Step := VISTEP_CREATE_DIR;
			ELSIF gVisionImage.CMD.DeleteDir THEN // Delete image directory on user partition including all images
				gVisionImage.DAT.Status := ERR_FUB_BUSY;
				Step := VISTEP_DELETE_DIR;
			ELSIF gVisionImage.CMD.DeleteImage THEN // Delete one image from the image directory on the user partition
				IF brsstrlen(ADR(visSelectedImage)) > 0 THEN
					brsstrcpy(ADR(FileNameComplete), ADR(gVisionImage.CFG.DirName));
					brsstrcat(ADR(FileNameComplete), ADR('/'));
					brsstrcat(ADR(FileNameComplete), ADR(visSelectedImage));
					gVisionImage.DAT.Status := ERR_FUB_BUSY;
					Step := VISTEP_DELETE_IMAGE;
				ELSE // No image selected --> do nothing, just reset the cmd
					gVisionImage.CMD.DeleteImage := FALSE;
				END_IF
			ELSIF gVisionImage.CMD.Refresh THEN // Refresh image list from the image directory on the user partition
				gVisionImage.DAT.Status := ERR_FUB_BUSY;
				Step := VISTEP_REFRESH_IMG_LIST;
			ELSIF gVisionImage.CMD.DownloadImage THEN // Download image from plc to webbrowser
				IF brsstrlen(ADR(visSelectedImage)) > 0 THEN
					brsstrcpy(ADR(FileNameComplete), ADR(gVisionImage.CFG.DirName));
					brsstrcat(ADR(FileNameComplete), ADR('/'));
					brsstrcat(ADR(FileNameComplete), ADR(visSelectedImage));
					gVisionImage.DAT.Status := ERR_FUB_BUSY;
					Step := VISTEP_DOWNLOAD_IMAGE;
				ELSE // If no pictures are available, don't try to download pictures
					gVisionImage.CMD.DownloadImage := FALSE;
				END_IF
			ELSIF gVisionImage.CMD.SaveImageOnPLC THEN // Save image from camera to PLC
				IF NOT gVisionImage.CFG.UploadBmpJpg AND NOT gVisionImage.CFG.UploadSVG THEN // Do nothing, because of no picture is needed
					gVisionImage.CMD.SaveImageOnPLC := FALSE;
					gVisionImage.DAT.Status	:= ERR_CFG_IMG;
				ELSIF gVisionSensor[LIMIT(1, gSelectedSensor, MAX_NUM_CAMS)].CFG.PowerlinkNode = 0 THEN
					gVisionImage.CMD.SaveImageOnPLC := FALSE;
					gVisionImage.DAT.Status	:= ERR_CFG_PLK;
				ELSE
					gVisionImage.DAT.Status	:= ERR_FUB_BUSY;
					Step := VISTEP_SAVE_IMG_ON_PLC;
				END_IF
			ELSIF gVisionImage.CMD.ResetError THEN // Reset error
				gVisionImage.CMD.ResetError := FALSE; // no error, so do nothing else (in case of an error, Step is VISTEP_ERR
			END_IF

			// Load new image into window
			IF visSelectedImageOld <> visSelectedImage AND ViRefreshImageList_0.DirEntries > 0 THEN
				brsmemset(ADR(visImagePath), 0, SIZEOF(visImagePath));
				visImagePath := '/FileDevice:';
				brsstrcat(ADR(visImagePath), ADR(gVisionImage.CFG.FileDevice));
				brsstrcat(ADR(visImagePath), ADR('/'));
				brsstrcat(ADR(visImagePath), ADR(gVisionImage.CFG.DirName));
				brsstrcat(ADR(visImagePath), ADR('/'));
				brsstrcat(ADR(visImagePath), ADR(visSelectedImage));
			ELSIF ViRefreshImageList_0.DirEntries = 0 THEN
				brsmemset(ADR(visImagePath), 0, SIZEOF(visImagePath));
			END_IF
			visSelectedImageOld := visSelectedImage;

			visEnableButtons_1 := Step = VISTEP_WAIT; // Disable buttons when command is pending: Save, Refresh, DeleteAll
			visEnableButtons_2 := visEnableButtons_1 AND ViRefreshImageList_0.DirEntries > 0 AND Step = VISTEP_WAIT; // Enable DeleteOneImage and DownloadImage button in mappView when no

		VISTEP_CREATE_DIR: // Create the image directory on user partition (if it does not exist)
			DirCreate_0.enable		:= TRUE;
			DirCreate_0.pDevice		:= ADR(gVisionImage.CFG.FileDevice);
			DirCreate_0.pName		:= ADR(gVisionImage.CFG.DirName);
			DirCreate_0();
			IF DirCreate_0.status = ERR_OK OR DirCreate_0.status = fiERR_DIR_ALREADY_EXIST THEN
				gVisionImage.CMD.CreateDir := FALSE;
				gVisionImage.CMD.DeleteDir := FALSE;
				gVisionImage.DAT.Status := 0;
				Step := VISTEP_REFRESH_IMG_LIST;
			ELSIF DirCreate_0.status <> ERR_FUB_BUSY THEN
				gVisionImage.DAT.Status := DirCreate_0.status;
				Step := VISTEP_ERR;
			END_IF

		VISTEP_DELETE_DIR: // Delete image directory on user partition including all images
			DirDeleteEx_0.enable	:= TRUE;
			DirDeleteEx_0.pDevice	:= ADR(gVisionImage.CFG.FileDevice);
			DirDeleteEx_0.pName		:= ADR(gVisionImage.CFG.DirName);
			DirDeleteEx_0();
			IF DirDeleteEx_0.status = ERR_OK THEN
				Step := VISTEP_CREATE_DIR;
			ELSIF DirDeleteEx_0.status <> ERR_FUB_BUSY THEN
				gVisionImage.DAT.Status := DirDeleteEx_0.status;
				Step := VISTEP_ERR;
			END_IF

		VISTEP_DELETE_IMAGE: // Delete one image from the image directory on the user partition
			FileDelete_0.enable 	:= TRUE;
			FileDelete_0.pDevice	:= ADR(gVisionImage.CFG.FileDevice);
			FileDelete_0.pName 		:= ADR(FileNameComplete);
			FileDelete_0();
			IF FileDelete_0.status = ERR_OK THEN
				gVisionImage.CMD.DeleteImage := FALSE;
				gVisionImage.DAT.Status := 0;
				Step := VISTEP_REFRESH_IMG_LIST;
			ELSIF FileDelete_0.status <> ERR_FUB_BUSY THEN
				gVisionImage.DAT.Status := FileDelete_0.status;
				Step := VISTEP_ERR;
			END_IF

		VISTEP_REFRESH_IMG_LIST: // Refresh image list from the image directory on the user partition
			ViRefreshImageList_0.Enable				:= TRUE;
			ViRefreshImageList_0.VisionImage		:= ADR(gVisionImage);
			ViRefreshImageList_0.ImageList			:= ADR(visImageList);
			ViRefreshImageList_0.visSelectedImage	:= ADR(visSelectedImage);
			ViRefreshImageList_0();
			IF ViRefreshImageList_0.Status = ERR_OK THEN
				gVisionImage.CMD.Refresh := FALSE;
				gVisionImage.DAT.Status := 0;
				Step := VISTEP_WAIT;
			ELSIF ViRefreshImageList_0.Status <> ERR_FUB_BUSY THEN
				gVisionImage.DAT.Status := ViRefreshImageList_0.Status;
				Step := VISTEP_ERR;
			END_IF

		VISTEP_DOWNLOAD_IMAGE: // Download image from plc to webbrowser
			ViDownloadImage_0.Enable				:= TRUE;
			ViDownloadImage_0.FileDevice			:= gVisionImage.CFG.FileDevice;
			ViDownloadImage_0.FileName				:= FileNameComplete;
			ViDownloadImage_0.ImgName				:= visSelectedImage;
			ViDownloadImage_0.visDownloadFileUrl	:= ADR(visDownloadFileUrl);
			ViDownloadImage_0();
			IF ViDownloadImage_0.Status = ERR_OK THEN
				gVisionImage.CMD.DownloadImage := FALSE;
				gVisionImage.DAT.Status := 0;
				Step := VISTEP_WAIT;
			ELSIF ViDownloadImage_0.Status <> ERR_FUB_BUSY THEN
				gVisionImage.DAT.Status := ViDownloadImage_0.Status;
				Step := VISTEP_ERR;
			END_IF

		VISTEP_SAVE_IMG_ON_PLC: // Save image from camera to PLC
			ViSaveImgOnPlc_0.Enable				:= TRUE;
			ViSaveImgOnPlc_0.CFG				:= gVisionImage.CFG;
			ViSaveImgOnPlc_0.PowerlinkNode		:= gVisionSensor[LIMIT(1, gSelectedSensor, MAX_NUM_CAMS)].CFG.PowerlinkNode;
			ViSaveImgOnPlc_0.CrossHairInfo		:= ADR(ViDrawCrosshair_0.CrossHairInfo);
			ViSaveImgOnPlc_0();
			IF ViSaveImgOnPlc_0.Status = ERR_OK THEN
				gVisionImage.CMD.SaveImageOnPLC := FALSE;
				gVisionImage.DAT.Status := 0;
				Step := VISTEP_REFRESH_IMG_LIST;
			ELSIF ViSaveImgOnPlc_0.Status <> ERR_FUB_BUSY THEN
				gVisionImage.DAT.Status := ViSaveImgOnPlc_0.Status;
				Step := VISTEP_ERR;
			END_IF

		VISTEP_ERR: // Error state
			IF gVisionImage.CMD.ResetError THEN
				gVisionImage.CMD.ResetError := FALSE;
				gVisionImage.DAT.Status := 0;
				Step := VISTEP_WAIT;
			END_IF
			brsmemset(ADR(gVisionImage.CMD), 0, SIZEOF(gVisionImage.CMD));
	END_CASE

	// Proxy server cyclic call ( Only needed for information. )
	ipSTR := gVisionImage.CFG.PlkIPWithoutNode;
	brsitoa(gSelectedSensor, ADR(nodeSTR));
	brsstrcat(ADR(ipSTR), ADR(nodeSTR));
	IF brsstrcmp( ADR( TcpForward_0.ConnectToIp ),ADR( ipSTR )) <> 0 THEN
		TcpForward_0.ConnectToIp := ipSTR ;
		TcpForward_0.Enable := FALSE ;
	ELSE
		TcpForward_0.Enable := gVisionSensor[gSelectedSensor].HW.Connected ; // Only enable if its connected
	END_IF
	TcpForward_0();

	// Draw the crosshairs on the mainpage
	ViDrawCrosshair_0.SelectedSensor		:= gSelectedSensor;
	ViDrawCrosshair_0.CmdRefreshCrosshair	:= gVisionImage.CMD.RefreshCrosshair;
	ViDrawCrosshair_0.VisionSensor			:= ADR(gVisionSensor[gSelectedSensor]);
	ViDrawCrosshair_0.CodeTypes				:= ADR(CodeTypes);
	ViDrawCrosshair_0.VisionDisabled		:= gVisionImage.DAT.VisionDisabled;
	ViDrawCrosshair_0.ImageRotation_deg		:= gVisionImage.CFG.ImageRotation_deg;
	ViDrawCrosshair_0.TextAlignment			:= visTextAlignment;
	ViDrawCrosshair_0.visCrossHair			:= ADR(visCrossHair);
	ViDrawCrosshair_0();
	gVisionImage.CMD.RefreshCrosshair		:= FALSE;

	// Create directory and files for showing the images on the mainpage in mappview visu
	IF NOT ViCreateWebDirFile_0.Done THEN
		ViCreateWebDirFile_0.Enable				:= TRUE;
		ViCreateWebDirFile_0.FileDevUser		:= gVisionImage.CFG.FileDevice;
		ViCreateWebDirFile_0.EthDevice			:= gVisionImage.CFG.EthDevice;
		ViCreateWebDirFile_0.EthIP				:= gVisionImage.CFG.EthIP;
		ViCreateWebDirFile_0.visWebViewerPath	:= ADR(visWebViewerPath);
		ViCreateWebDirFile_0();
	END_IF
	visWebViewerQuery := 'q=';
	brsitoa(gVisionImage.CFG.MainPageQualityJPG, ADR(tmpStr));
	brsstrcat(ADR(visWebViewerQuery), ADR(tmpStr));
	brsstrcat(ADR(visWebViewerQuery), ADR('&rot='));
	brsitoa(gVisionImage.CFG.ImageRotation_deg, ADR(tmpStr));
	brsstrcat(ADR(visWebViewerQuery), ADR(tmpStr));
	brsstrcat(ADR(visWebViewerQuery), ADR('&scale='));
	CASE gVisionImage.CFG.ImageRotation_deg OF
		0:		brsftoa(1.0, ADR(tmpStr));
		90:		brsftoa(UINT_TO_REAL(gVisionSensor[gSelectedSensor].CFG.ResolutionHeight_Y) / UINT_TO_REAL(gVisionSensor[gSelectedSensor].CFG.ResolutionWidth_X), ADR(tmpStr));
		180:	brsftoa(1.0, ADR(tmpStr));
		270:	brsftoa(UINT_TO_REAL(gVisionSensor[gSelectedSensor].CFG.ResolutionHeight_Y) / UINT_TO_REAL(gVisionSensor[gSelectedSensor].CFG.ResolutionWidth_X), ADR(tmpStr));
	ELSE
		brsftoa(1.0, ADR(tmpStr));
	END_CASE
	brsstrcat(ADR(visWebViewerQuery), ADR(tmpStr));

	// Main page image rotation
	gVisionImage.CFG.ImageRotation_deg := visImageRotation * 90;

	// Show camera image on VC4 visualization
	ViShowImgOnVC4_0.Enable				:= ViCreateWebDirFile_0.Done; // Wait until the directory "web" is created
	ViShowImgOnVC4_0.RefreshImage		:= visVC4RefreshImg;
	ViShowImgOnVC4_0.CFG				:= gVisionImage.CFG;
	ViShowImgOnVC4_0.PowerlinkNode		:= gVisionSensor[LIMIT(1, gSelectedSensor, MAX_NUM_CAMS)].CFG.PowerlinkNode;
	ViShowImgOnVC4_0.ImgWidthInVC4_px	:= 500; // Pixel
	ViShowImgOnVC4_0();
	IF ViShowImgOnVC4_0.RefreshDone THEN
		visVC4RefreshImg := FALSE;
	END_IF

	// Refreh crosshairs when new image is available
	IF EDGENEG(gVisionSensor[gSelectedSensor].CMD.ImageTrigger) THEN
		gVisionImage.CMD.RefreshCrosshair := TRUE;
	END_IF
	gVisionImage.DAT.VisionDisabled := NOT gVisionSensor[gSelectedSensor].DAT.Enable;

	brsmemcpy(ADR(RemCfgImage), ADR(gVisionImage.CFG), SIZEOF(RemCfgImage)); // Save settings to remanent variable
END_PROGRAM
PROGRAM _EXIT
	(* After download make sure to close this connection. If this is not closed the functionblock cant retrieve the new information *)
	TcpForward_0.Enable := FALSE;
	TcpForward_0();
END_PROGRAM
```

#### ViCreateWebDirFile.st
```iecst
FUNCTION_BLOCK ViCreateWebDirFile
	IF NOT Enable THEN
		Status := ERR_FUB_ENABLE_FALSE;
		Step := 0;
		RETURN;
	END_IF
	CASE Step OF
		0:
			Status := ERR_FUB_BUSY;
			Done := FALSE;
			Step := 1;
		1: // Init
			ACTION_CreateHtmlFile;
			FileDevSystem		:= 'CF';
			FileDevSystemPara	:= '/DEVICE=C:/';
			DirNameWeb			:= 'web';
			FileNameVisImgHtml	:= 'web/VisionImg.html';
			FileNameEyeSystem	:= 'ADDONS/DATA/IAT_Data/wwwRoot/BRVisu/Media/VisionEye.png';
			FileNameEyeUser		:= 'web/VisionEye.png';
			Step := 2;
		2: // Check if web directory already exists
			DirInfo_0(enable := TRUE, pDevice := ADR(FileDevUser), pPath := ADR(DirNameWeb));
			IF DirInfo_0.status = ERR_OK THEN
				Step := 9;
			ELSIF DirInfo_0.status = fiERR_DIR_NOT_EXIST THEN
				Step := 3;
			ELSIF DirInfo_0.status <> ERR_FUB_BUSY THEN
				Status := DirInfo_0.status;
				Step := 0;
			END_IF
		3: // Create web directory if it does not exist
			DirCreate_0(enable := TRUE, pDevice := ADR(FileDevUser), pName := ADR(DirNameWeb));
			IF DirCreate_0.status = ERR_OK THEN
				Step := 10;
			ELSIF DirCreate_0.status <> ERR_FUB_BUSY THEN
				Status := DirCreate_0.status;
				Step := 0;
			END_IF
		9: // Try to delete the html file. This is necessary, because of when settings are changed, the file needs to be recreated.
			FileDelete_0(enable := TRUE, pDevice := ADR(FileDevUser), pName := ADR(FileNameVisImgHtml));
			IF FileDelete_0.status = ERR_OK OR FileDelete_0.status = fiERR_FILE_NOT_FOUND THEN
				Step := 10;
			ELSIF FileDelete_0.status <> ERR_FUB_BUSY THEN
				Status := FileDelete_0.status;
				Step := 0;
			END_IF
		10: // Check if html page exists
			FileCreate_0(enable := TRUE, pDevice := ADR(FileDevUser), pFile := ADR(FileNameVisImgHtml));
			IF FileCreate_0.status = ERR_OK THEN
				brsstrcpy(ADR(FileWriteData), ADR(HtmlFileContent1));
				brsstrcat(ADR(FileWriteData), ADR(EthIP));
				brsstrcat(ADR(FileWriteData), ADR(HtmlFileContent2));
				Step := 11;
			ELSIF FileCreate_0.status = fiERR_EXIST THEN
				Step := 20;
			ELSIF FileCreate_0.status <> ERR_FUB_BUSY THEN
				Status := FileCreate_0.status;
				Step := 0;
			END_IF
		11: // Write content
			FileWrite_0(enable := TRUE, ident := FileCreate_0.ident, offset := 0, pSrc := ADR(FileWriteData), len := brsstrlen(ADR(FileWriteData)));
			IF FileWrite_0.status = ERR_OK THEN
				Step := 12;
			ELSIF FileWrite_0.status <> ERR_FUB_BUSY THEN
				Status := FileWrite_0.status;
				Step := 0;
			END_IF
		12: // Close file
			FileClose_0(enable := TRUE, ident := FileCreate_0.ident);
			IF FileClose_0.status = ERR_OK THEN
				Step := 20;
			ELSIF FileClose_0.status <> ERR_FUB_BUSY THEN
				Status := FileClose_0.status;
				Step := 0;
			END_IF

		20: // Create FileDevice to System partition
			DevLink_0(enable := TRUE, pDevice := ADR(FileDevSystem), pParam := ADR(FileDevSystemPara));
			IF DevLink_0.status = ERR_OK THEN
				Step := 21;
			ELSIF DevLink_0.status <> ERR_FUB_BUSY THEN
				Status := DevLink_0.status;
				Step := 0;
			END_IF
		21: // Copy VisionEye.png from mappView folder (System partition) to webserver dir
			FileCopy_0(enable := TRUE, pSrcDev := ADR(FileDevSystem), pSrc := ADR(FileNameEyeSystem), pDestDev := ADR(FileDevUser), pDest := ADR(FileNameEyeUser));
			IF FileCopy_0.status <> ERR_FUB_BUSY THEN
				Status := FileCopy_0.status;
				Step := 22;
			END_IF
		22: // Delete DevLink
			DevUnlink_0(enable := TRUE, handle := DevLink_0.handle);
			IF DevUnlink_0.status = ERR_OK THEN
				Step := 30;
			ELSIF DevUnlink_0.status <> ERR_FUB_BUSY THEN
				Status := DevUnlink_0.status;
				Step := 0;
			END_IF
		30: // Create path for webviewer widget
			visWebViewerPath := 'http://'; // Create path for webviewer widget
			brsstrcat(ADR(visWebViewerPath), ADR(EthIP));
			Done := TRUE;
			Status := ERR_OK;
			Step := 0;
	END_CASE
END_FUNCTION_BLOCK
```

#### ViDrawCrosshair.st
```iecst
FUNCTION_BLOCK ViDrawCrosshair
	// Assign pointers
	IF VisionSensor.CFG.DataStructure <> 0 THEN
		CASE VisionSensor.CFG.VisionFunction OF
			enumBlob:
				Blob ACCESS VisionSensor.CFG.DataStructure;
			enumCoderReader:
				CodeReader ACCESS VisionSensor.CFG.DataStructure;
			enumMatch:
				Match ACCESS VisionSensor.CFG.DataStructure;
			enumMeasurement:
				MT ACCESS VisionSensor.CFG.DataStructure;
			enumOCR:
				OCR ACCESS VisionSensor.CFG.DataStructure;
			enumPixelCounter:
				Pixel ACCESS VisionSensor.CFG.DataStructure;
		END_CASE
	ELSE
		RETURN;
	END_IF

	// Draw cross hairs
	IF CmdRefreshCrosshair OR (visCrossHair.ShowCrosshair <> ShowCrosshairOld) OR (visCrossHair.DetailsNo <> DetailsNoOld) OR (SelectedSensor <> SelectedSensorOld) OR (ImageRotation_deg <> ImageRotation_degOld) OR (TextAlignment <> TextAlignmentOld) THEN
		ShowCrosshairOld		:= visCrossHair.ShowCrosshair;
		SelectedSensorOld		:= SelectedSensor;
		ImageRotation_degOld	:= ImageRotation_deg;
		TextAlignmentOld		:= TextAlignment;
		// First delete transformation and make everything invisible
		brsmemset(ADR(visCrossHair.SvgTransformation), 0, SIZEOF(visCrossHair.SvgTransformation));
		brsmemset(ADR(visCrossHair.SvgVisible), 0, SIZEOF(visCrossHair.SvgVisible));
		IF visCrossHair.ShowCrosshair THEN
			// Handle details no
			IF visCrossHair.DetailsNo < 1 THEN
				IF VisionSensor.DAT.ResultCnt > 0 THEN
					visCrossHair.DetailsNo := VisionSensor.DAT.ResultCnt;
				ELSE
					visCrossHair.DetailsNo := 1;
				END_IF
			END_IF
			IF visCrossHair.DetailsNo > VisionSensor.DAT.ResultCnt THEN
				visCrossHair.DetailsNo := 1;
			END_IF
			DetailsNoOld := visCrossHair.DetailsNo;

			// Create cross hairs and data for all results
			FOR idx := 1 TO MAX_NUM_RESULTS DO
				ResultModelNumber	:= 0;
				ResultPositionX		:= 0;
				ResultPositionY		:= 0;
				ResultOrientation	:= 0;
				brsmemset(ADR(CrossHairInfo[idx]), 0, SIZEOF(CrossHairInfo[0]));

				// Make sure we have data to display
				IF VisionSensor.DAT.ResultCnt <> 0 AND idx <= VisionSensor.DAT.ResultCnt THEN
					// Select data source from vision function
					MT_UseXY := FALSE;
					CASE VisionSensor.CFG.VisionFunction OF
						enumBlob:
							ResultModelNumber	:= Blob.ModelNumber[idx];
							ResultPositionX		:= UDINT_TO_REAL(Blob.PositionX[idx]) / visCrossHair.CFG.PixelRatio;
							ResultPositionY		:= UDINT_TO_REAL(Blob.PositionY[idx]) / visCrossHair.CFG.PixelRatio;
							ResultOrientation	:= Blob.Orientation[idx] / visCrossHair.CFG.PixelRatio;
						enumPixelCounter:
							ResultModelNumber	:= Pixel.ModelNumber[idx];
							ResultPositionX		:= UDINT_TO_REAL(Pixel.PositionX[idx]) / visCrossHair.CFG.PixelRatio;
							ResultPositionY		:= UDINT_TO_REAL(Pixel.PositionY[idx]) / visCrossHair.CFG.PixelRatio;
						enumCoderReader:
							ResultPositionX		:= UDINT_TO_REAL(CodeReader.PositionX[idx]) / visCrossHair.CFG.PixelRatio;
							ResultPositionY		:= UDINT_TO_REAL(CodeReader.PositionY[idx]) / visCrossHair.CFG.PixelRatio;
							ResultOrientation	:= CodeReader.Orientation[idx] / visCrossHair.CFG.PixelRatio;
						enumMatch:
							ResultModelNumber	:= Match.ModelNumber[idx];
							ResultPositionX		:= UDINT_TO_REAL(Match.PositionX[idx]) / visCrossHair.CFG.PixelRatio;
							ResultPositionY		:= UDINT_TO_REAL(Match.PositionY[idx]) / visCrossHair.CFG.PixelRatio;
							ResultOrientation	:= Match.Orientation[idx] / visCrossHair.CFG.PixelRatio;
						enumMeasurement:
							IF MT.UseResultAsXY THEN
								ResultPositionX	:= UDINT_TO_REAL(MT.Result[idx])/10;
								ResultPositionY	:= UDINT_TO_REAL(MT.Result[idx+1])/10;
								idx := idx + 1;
							END_IF
							MT_UseXY := TRUE; // use this variable because of in case Visionfunction != MT then the Pointer MT is not initialized
						enumOCR:
							ResultPositionX		:= UDINT_TO_REAL(OCR.PositionX[idx]) / visCrossHair.CFG.PixelRatio;
							ResultPositionY		:= UDINT_TO_REAL(OCR.PositionY[idx]) / visCrossHair.CFG.PixelRatio;
							ResultOrientation	:= OCR.Orientation[idx] / visCrossHair.CFG.PixelRatio;
					END_CASE

					// Adapt the size to the size of the WebViewer image in mapp View. The download as svg file also uses a fixed size (both 1280x1024)
					ResultPositionX				:= ResultPositionX * UINT_TO_REAL(visCrossHair.CFG.RefSizeX) / UINT_TO_REAL(VisionSensor.CFG.ResolutionWidth_X);
					ResultPositionY				:= ResultPositionY * UINT_TO_REAL(visCrossHair.CFG.RefSizeY) / UINT_TO_REAL(VisionSensor.CFG.ResolutionHeight_Y);

					// Show crosshair except for measurement function
					IF VisionSensor.CFG.VisionFunction <> enumMeasurement OR MT_UseXY THEN
						IF ResultPositionX <> 0 AND ResultPositionY <> 0 THEN
							visCrossHair.SvgVisible[idx] := TRUE;

							// Calculate cross information, also needed for saving the svg in ViSaveImgOnPLC
							CrossHairInfo[idx].CrosshairScale			:= visCrossHair.CFG.Scale;
							CrossHairInfo[idx].CrosshairSizeScaled		:= USINT_TO_REAL(visCrossHair.CFG.Size) * visCrossHair.CFG.Scale;
							CrossHairInfo[idx].CrosshairTopLeftX		:= ResultPositionX - CrossHairInfo[idx].CrosshairSizeScaled / 2.0;
							CrossHairInfo[idx].CrosshairTopLeftY		:= ResultPositionY - CrossHairInfo[idx].CrosshairSizeScaled / 2.0;
							CrossHairInfo[idx].CrosshairRotateCenter	:= ResultOrientation * -1;

							// Crosshair transformation for displaying in the mappView visu
							IF visCrossHair.DetailsNo = idx THEN
								svgTrafo := '[{"select":"#CrosshairBlue","display":false}, {"select":"#CrosshairRed","display":true, "translate":[';
							ELSE
								svgTrafo := '[{"select":"#CrosshairRed","display":false}, { "select":"#CrosshairBlue","display":true, "translate":[';
							END_IF
							// Crosshair position
							CrosshSize		:= CrossHairInfo[idx].CrosshairSizeScaled / 2.0;
							ScaleVertical	:= UINT_TO_REAL(VisionSensor.CFG.ResolutionHeight_Y) / UINT_TO_REAL(VisionSensor.CFG.ResolutionWidth_X);
							CASE ImageRotation_deg OF
								0:		brsitoa(REAL_TO_INT(ResultPositionX															- CrosshSize), ADR(tmpStr));
								90:		brsitoa(REAL_TO_INT((VisionSensor.CFG.ResolutionHeight_Y - ResultPositionY) * ScaleVertical	- CrosshSize), ADR(tmpStr));
								180:	brsitoa(REAL_TO_INT(VisionSensor.CFG.ResolutionWidth_X - ResultPositionX					- CrosshSize), ADR(tmpStr));
								270:	brsitoa(REAL_TO_INT(ResultPositionY * ScaleVertical											- CrosshSize), ADR(tmpStr));
							ELSE
										brsitoa(REAL_TO_INT(ResultPositionX															- CrosshSize), ADR(tmpStr));
							END_CASE
							brsstrcat(ADR(svgTrafo), ADR(tmpStr));
							brsstrcat(ADR(svgTrafo), ADR(','));
							CASE ImageRotation_deg OF
								0:		brsitoa(REAL_TO_INT(ResultPositionY															- CrosshSize), ADR(tmpStr));
								90:		brsitoa(REAL_TO_INT(ResultPositionX * ScaleVertical											- CrosshSize), ADR(tmpStr));
								180:	brsitoa(REAL_TO_INT(VisionSensor.CFG.ResolutionHeight_Y - ResultPositionY					- CrosshSize), ADR(tmpStr));
								270:	brsitoa(REAL_TO_INT((VisionSensor.CFG.ResolutionWidth_X - ResultPositionX) * ScaleVertical	- CrosshSize), ADR(tmpStr));
							ELSE
										brsitoa(REAL_TO_INT(ResultPositionY															- CrosshSize), ADR(tmpStr));
							END_CASE
							brsstrcat(ADR(svgTrafo), ADR(tmpStr));
							// Add cross hair scaling
							brsstrcat(ADR(svgTrafo), ADR('],"scale":['));
							brsftoa(visCrossHair.CFG.Scale, ADR(tmpStr));
							brsstrcat(ADR(svgTrafo), ADR(tmpStr));
							brsstrcat(ADR(svgTrafo), ADR(','));
							brsstrcat(ADR(svgTrafo), ADR(tmpStr));
							// Add cross hair rotation
							brsstrcat(ADR(svgTrafo), ADR('],"spin":['));
							brsftoa(CrossHairInfo[idx].CrosshairRotateCenter - ImageRotation_deg, ADR(tmpStr));
							brsstrcat(ADR(svgTrafo), ADR(tmpStr));
							brsstrcat(ADR(svgTrafo), ADR(','));
							brsftoa(USINT_TO_REAL(visCrossHair.CFG.Size) / 2, ADR(tmpStr)); // For mappView the rotation is based on the original size, not on the scaled size
							brsstrcat(ADR(svgTrafo), ADR(tmpStr));
							brsstrcat(ADR(svgTrafo), ADR(','));
							brsstrcat(ADR(svgTrafo), ADR(tmpStr));
							brsstrcat(ADR(svgTrafo), ADR(']}]'));
							visCrossHair.SvgTransformation[idx] := svgTrafo;

							// Add text data to selected cross hair (small index number)
							IF visCrossHair.DetailsNo = idx THEN
								svgContent := '<text class="cText" fill="red " font-size="22" font-family="Helvetica, Arial, sans-serif"><tspan class="text" x="';
							ELSE
								svgContent := '<text class="cText" fill="blue" font-size="22" font-family="Helvetica, Arial, sans-serif"><tspan class="text" x="';
							END_IF
							CASE ImageRotation_deg OF
								0:		brsitoa(REAL_TO_INT(ResultPositionX															+ CrosshSize), ADR(tmpStr));
								90:		brsitoa(REAL_TO_INT((VisionSensor.CFG.ResolutionHeight_Y - ResultPositionY) * ScaleVertical	+ CrosshSize), ADR(tmpStr));
								180:	brsitoa(REAL_TO_INT(VisionSensor.CFG.ResolutionWidth_X - ResultPositionX					+ CrosshSize), ADR(tmpStr));
								270:	brsitoa(REAL_TO_INT(ResultPositionY * ScaleVertical											+ CrosshSize), ADR(tmpStr));
							ELSE
										brsitoa(REAL_TO_INT(ResultPositionX															+ CrosshSize), ADR(tmpStr));
							END_CASE
							brsstrcat(ADR(svgContent), ADR(tmpStr));
							brsstrcat(ADR(svgContent), ADR('" y="'));
							CASE ImageRotation_deg OF
								0:		brsitoa(REAL_TO_INT(ResultPositionY															+ 5), ADR(tmpStr));
								90:		brsitoa(REAL_TO_INT(ResultPositionX * ScaleVertical											+ 5), ADR(tmpStr));
								180:	brsitoa(REAL_TO_INT(VisionSensor.CFG.ResolutionHeight_Y - ResultPositionY					+ 5), ADR(tmpStr));
								270:	brsitoa(REAL_TO_INT((VisionSensor.CFG.ResolutionWidth_X - ResultPositionX) * ScaleVertical	+ 5), ADR(tmpStr));
							ELSE
										brsitoa(REAL_TO_INT(ResultPositionY															+ 5), ADR(tmpStr));
							END_CASE
							brsstrcat(ADR(svgContent), ADR(tmpStr));
							brsstrcat(ADR(svgContent), ADR('"> '));
							// Add result number
							brsitoa(idx, ADR(tmpStr));
							brsstrcat(ADR(svgContent), ADR(tmpStr));
							brsstrcat(ADR(svgContent), ADR('</tspan></text>'));

							// for saving svg file. The texts added below are not of interest for the saved SVG, so copy it now before adding the details information
							brsstrcpy(ADR(CrossHairInfo[idx].Text), ADR(svgContent));
							blueTextPos := FIND(CrossHairInfo[idx].Text, 'fill="blue"'); // Make all texts red. In the SVG is no highlighted crosshair
							IF blueTextPos > 2 THEN
								brsmemcpy(ADR(CrossHairInfo[idx].Text) + blueTextPos - 1, ADR('fill="red "'), 11);
							END_IF
							visCrossHair.SvgContent[idx] := svgContent;

							// Create details information to show in the top left or right corner
							brsstrcat(ADR(svgContent), ADR('<text class="cText" fill="red" font-size="35" font-family="Helvetica, Arial, sans-serif" x="10" y="10"> '));
							CrossHairInfo[1].DataVis	:= '';
							CrossHairInfo[idx].Data		:= '';
							// Add model ID information for blob and match
							IF VisionSensor.CFG.VisionFunction = enumBlob OR VisionSensor.CFG.VisionFunction = enumMatch THEN
								CrosshairDetailsValue(ADR(svgContent),  ADR('Model ID: '), ResultModelNumber, TextAlignment);
								brsstrcat(ADR(CrossHairInfo[1].DataVis), ADR('1, '));
								brsitoa(ResultModelNumber, ADR(tmpStr));
								brsstrcat(ADR(CrossHairInfo[idx].Data), ADR(tmpStr));
								brsstrcat(ADR(CrossHairInfo[idx].Data), ADR(', '));
							ELSE
								brsstrcat(ADR(CrossHairInfo[1].DataVis), ADR('0, '));
								brsstrcat(ADR(CrossHairInfo[idx].Data), ADR('"none", '));
							END_IF
							// Add X and Y position information
							CrosshairDetailsValue(ADR(svgContent),  ADR('Pos X: '), ResultPositionX, TextAlignment);
							CrosshairDetailsValue(ADR(svgContent),  ADR('Pos Y: '), ResultPositionY, TextAlignment);
							brsstrcat(ADR(CrossHairInfo[1].DataVis), ADR('1, 1, '));
							brsftoa(ResultPositionX, ADR(tmpStr));
							brsstrcat(ADR(CrossHairInfo[idx].Data), ADR(tmpStr));
							brsstrcat(ADR(CrossHairInfo[idx].Data), ADR(', '));
							brsftoa(ResultPositionY, ADR(tmpStr));
							brsstrcat(ADR(CrossHairInfo[idx].Data), ADR(tmpStr));
							brsstrcat(ADR(CrossHairInfo[idx].Data), ADR(', '));
							// Add orientation information
							IF VisionSensor.CFG.VisionFunction <> enumMeasurement THEN
								CrosshairDetailsValue(ADR(svgContent),  ADR('Orientation: '), ResultOrientation, TextAlignment);
								brsstrcat(ADR(CrossHairInfo[1].DataVis), ADR('1, '));
								brsftoa(ResultOrientation, ADR(tmpStr));
								brsstrcat(ADR(CrossHairInfo[idx].Data), ADR(tmpStr));
								brsstrcat(ADR(CrossHairInfo[idx].Data), ADR(', '));
							ELSE
								brsstrcat(ADR(CrossHairInfo[1].DataVis), ADR('0, '));
								brsstrcat(ADR(CrossHairInfo[idx].Data), ADR('"none", '));
							END_IF
							// Add detail information for blob
							IF VisionSensor.CFG.VisionFunction = enumBlob THEN
								IF Blob.EnhancedBlobInformation = 1 THEN // Only access the Pointer Blob if it really exists. So don't combine this line of code with the line before
									CrosshairDetailsValue(ADR(svgContent),  ADR('Clipped: '), Blob.Clipped[idx], TextAlignment);
									CrosshairDetailsValue(ADR(svgContent),  ADR('Gray: '), Blob.MeanGrayValue[idx], TextAlignment);
									CrosshairDetailsValue(ADR(svgContent),  ADR('Length: '), UDINT_TO_REAL(Blob.Length[idx])/visCrossHair.CFG.PixelRatio, TextAlignment);
									CrosshairDetailsValue(ADR(svgContent),  ADR('Width: '), UDINT_TO_REAL(Blob.Width[idx])/visCrossHair.CFG.PixelRatio, TextAlignment);
									CrosshairDetailsValue(ADR(svgContent),  ADR('Area: '), UDINT_TO_REAL(Blob.Area[idx])/visCrossHair.CFG.PixelRatio, TextAlignment);
									brsstrcat(ADR(CrossHairInfo[1].DataVis), ADR('1, 1, 1, 1, 1, '));
									brsitoa(Blob.Clipped[idx], ADR(tmpStr));
									brsstrcat(ADR(CrossHairInfo[idx].Data), ADR(tmpStr));
									brsstrcat(ADR(CrossHairInfo[idx].Data), ADR(', '));
									brsitoa(Blob.MeanGrayValue[idx], ADR(tmpStr));
									brsstrcat(ADR(CrossHairInfo[idx].Data), ADR(tmpStr));
									brsstrcat(ADR(CrossHairInfo[idx].Data), ADR(', '));
									brsftoa(UDINT_TO_REAL(Blob.Length[idx])/visCrossHair.CFG.PixelRatio, ADR(tmpStr));
									brsstrcat(ADR(CrossHairInfo[idx].Data), ADR(tmpStr));
									brsstrcat(ADR(CrossHairInfo[idx].Data), ADR(', '));
									brsftoa(UDINT_TO_REAL(Blob.Width[idx])/visCrossHair.CFG.PixelRatio, ADR(tmpStr));
									brsstrcat(ADR(CrossHairInfo[idx].Data), ADR(tmpStr));
									brsstrcat(ADR(CrossHairInfo[idx].Data), ADR(', '));
									brsftoa(UDINT_TO_REAL(Blob.Area[idx])/visCrossHair.CFG.PixelRatio, ADR(tmpStr));
									brsstrcat(ADR(CrossHairInfo[idx].Data), ADR(tmpStr));
									brsstrcat(ADR(CrossHairInfo[idx].Data), ADR(', '));
								ELSE
									brsstrcat(ADR(CrossHairInfo[1].DataVis), ADR('0, 0, 0, 0, 0, '));
									brsstrcat(ADR(CrossHairInfo[idx].Data), ADR('"none", "none", "none", "none", "none", '));
								END_IF
							ELSE
								brsstrcat(ADR(CrossHairInfo[1].DataVis), ADR('0, 0, 0, 0, 0, '));
								brsstrcat(ADR(CrossHairInfo[idx].Data), ADR('"none", "none", "none", "none", "none", '));
							END_IF
							// Add detail information for match
							IF VisionSensor.CFG.VisionFunction = enumMatch THEN
								CrosshairDetailsValue(ADR(svgContent),  ADR('Score: '), Match.Score[idx], TextAlignment);
								CrosshairDetailsValue(ADR(svgContent),  ADR('Scale: '), Match.Scale[idx], TextAlignment);
								brsstrcat(ADR(CrossHairInfo[1].DataVis), ADR('1, 1, '));
								brsitoa(Match.Score[idx], ADR(tmpStr));
								brsstrcat(ADR(CrossHairInfo[idx].Data), ADR(tmpStr));
								brsstrcat(ADR(CrossHairInfo[idx].Data), ADR(', '));
								brsitoa(Match.Scale[idx], ADR(tmpStr));
								brsstrcat(ADR(CrossHairInfo[idx].Data), ADR(tmpStr));
								brsstrcat(ADR(CrossHairInfo[idx].Data), ADR(', '));
							ELSE
								brsstrcat(ADR(CrossHairInfo[1].DataVis), ADR('0, 0, '));
								brsstrcat(ADR(CrossHairInfo[idx].Data), ADR('"none", "none", '));
							END_IF
							// Add detail information for OCR and CodeReader
							IF VisionSensor.CFG.VisionFunction = enumOCR THEN
								CrosshairDetailsValue(ADR(svgContent),  ADR('Grading: '), OCR.Grading[idx], TextAlignment);
								CrosshairDetailsText(ADR(svgContent),  ADR('Text: '), ADR(OCR.Text[idx]), TextAlignment);
								brsstrcat(ADR(CrossHairInfo[1].DataVis), ADR('1, 0, 1, ')); // Grading, Code Type, Text
								brsitoa(OCR.Grading[idx], ADR(tmpStr));
								brsstrcat(ADR(CrossHairInfo[idx].Data), ADR(tmpStr));
								brsstrcat(ADR(CrossHairInfo[idx].Data), ADR(', "none", "'));
								brsstrcat(ADR(CrossHairInfo[idx].Data), ADR(OCR.Text[idx]));
								brsstrcat(ADR(CrossHairInfo[idx].Data), ADR('", '));
							ELSIF VisionSensor.CFG.VisionFunction = enumCoderReader THEN
								CrosshairDetailsText(ADR(svgContent),  ADR('Code: '), ADR(CodeTypes[LIMIT(0, CodeReader.BarcodeType[idx], MAX_NUM_CODETYPES)]), TextAlignment);
								CrosshairDetailsText(ADR(svgContent),  ADR('Text: '), ADR(CodeReader.BarcodeText[idx]), TextAlignment);
								brsstrcat(ADR(CrossHairInfo[1].DataVis), ADR('0, 1, 1, ')); // Grading, Code Type, Text
								brsstrcat(ADR(CrossHairInfo[idx].Data), ADR('"none", "'));
								brsstrcat(ADR(CrossHairInfo[idx].Data), ADR(CodeTypes[LIMIT(0, CodeReader.BarcodeType[idx], MAX_NUM_CODETYPES)]));
								brsstrcat(ADR(CrossHairInfo[idx].Data), ADR('", "'));
								brsstrcat(ADR(CrossHairInfo[idx].Data), ADR(CodeReader.BarcodeText[idx]));
								brsstrcat(ADR(CrossHairInfo[idx].Data), ADR('", '));
							ELSE
								brsstrcat(ADR(CrossHairInfo[1].DataVis), ADR('0, 0, 0, '));
								brsstrcat(ADR(CrossHairInfo[idx].Data), ADR('"none", "none", "none", '));
							END_IF
							brsstrcat(ADR(CrossHairInfo[1].DataVis), ADR('0')); // For the not used "Result"
							brsstrcat(ADR(CrossHairInfo[idx].Data), ADR('"none"')); // For the not used "Result"
							brsstrcat(ADR(svgContent), ADR('</text>'));
							// Add text data from selected cross hair in the top left corner of the image, but only if the index is the actual index
							IF visCrossHair.DetailsNo = idx THEN
								visCrossHair.SvgContent[idx] := svgContent;
							END_IF
						END_IF
					ELSE // Add result information for measurement
						visCrossHair.SvgTransformation[idx] := '[{"select":"#CrosshairRed","display":false}, {"select":"#CrosshairBlue","display":false}]';
						visCrossHair.SvgVisible[idx] := TRUE;
						brsstrcpy(ADR(svgContent), ADR('<text class="cText" fill="red" font-size="35" font-family="Helvetica, Arial, sans-serif" x="10" y="'));
						brsitoa(idx*40, ADR(tmpStr));
						brsstrcat(ADR(svgContent), ADR(tmpStr));
						brsstrcat(ADR(svgContent), ADR('"> '));
						CrosshairDetailsValue(ADR(svgContent),  ADR('Result:'), UDINT_TO_REAL(MT.Result[idx])/1000, TextAlignment);
						brsstrcat(ADR(svgContent), ADR('</text>'));
						visCrossHair.SvgContent[idx] := svgContent;
						brsstrcpy(ADR(CrossHairInfo[1].DataVis), ADR('0, 0, 0, 0, 0, 0, 0, 0, 0, 0, 0, 0, 0, 0, 1'));
						brsstrcpy(ADR(CrossHairInfo[idx].Data), ADR('"none", "none", "none", "none", "none", "none", "none", "none", "none", "none", "none", "none", "none", "none", '));
						brsftoa(UDINT_TO_REAL(MT.Result[idx])/1000, ADR(tmpStr));
						brsstrcat(ADR(CrossHairInfo[idx].Data), ADR(tmpStr));
					END_IF
				ELSIF VisionSensor.DAT.ResultCnt = 0 AND VisionDisabled THEN // Vision function is disabled --> show a message
					visCrossHair.SvgVisible[1]			:= TRUE;
					visCrossHair.SvgTransformation[1]	:= '[{"select":"#CrosshairRed","display":false}, {"select":"#CrosshairBlue","display":false}]';
					visCrossHair.SvgContent[1]			:= '<text class="cText" fill="red" font-size="35" font-family="Helvetica, Arial, sans-serif" x="10" y="40"> Processing is disabled </text>';
				END_IF
			END_FOR
		END_IF // IF visCrossHair.ShowCrosshair THEN
	END_IF
END_FUNCTION_BLOCK
```

### Library Logical/old/Vi_visu

#### Variables.var
```iecst
(*-----------------------------------------------------------------------------------------------------------------------------------------*)
(*Main vision and data structures*)
VAR
	VisionSensor : REFERENCE TO typVisionMain; (*General vision functions that are independent from the inspection function*)
	VisionLight : REFERENCE TO typLightMain; (*General vision functions that are independent from the inspection function*)
	Match : REFERENCE TO typMatchMain; (*Data that is specific for the match function*)
	CodeReader : REFERENCE TO typCodeReaderMain; (*Data that is specific for the code reader*)
	MT : REFERENCE TO typMTMain; (*Data that is specific for the MT function*)
	OCR : REFERENCE TO typOCRMain; (*Data that is specific for the OCR function*)
	Blob : REFERENCE TO typBlobMain; (*Data that is specific for the blob function*)
	Pixel : REFERENCE TO typPixelMain; (*Data that is specific for the blob function*)
	tmpMatch : {REDUND_UNREPLICABLE} typMatchMain; (*Data that is specific for the match function*)
	tmpCodeReader : {REDUND_UNREPLICABLE} typCodeReaderMain; (*Data that is specific for the code reader*)
	tmpMT : {REDUND_UNREPLICABLE} typMTMain; (*Data that is specific for the OCR function*)
	tmpOCR : {REDUND_UNREPLICABLE} typOCRMain; (*Data that is specific for the OCR function*)
	tmpBlob : {REDUND_UNREPLICABLE} typBlobMain; (*Data that is specific for the blob function*)
	tmpPixel : {REDUND_UNREPLICABLE} typPixelMain; (*Data that is specific for the blob function*)
END_VAR
(*-----------------------------------------------------------------------------------------------------------------------------------------*)
(*Vision function blocks*)
VAR
	VaGetList_01 : VaGetList;
END_VAR
(*-----------------------------------------------------------------------------------------------------------------------------------------*)
(*Sensor variables*)
VAR
	visAutoArchiv : BOOL;
	visSensorEnableCommand : BOOL; (*Enable/Disable vision trigger and enable when camera is not ready*)
	visEnableSetup : BOOL; (*Enable/Disable vision setup when camera is not ready*)
	visEnableRepetitive : BOOL; (*Enable/Disable repetitive mode*)
	visImageTrigger : BOOL; (*Trigger new image*)
	visVisionApplicationList : ARRAY[0..19] OF STRING[80]; (*Flash color string*)
	visSensorFlashColor : STRING[10]; (*Flash color string*)
	visSensorFlashColorOld : STRING[10]; (*Flash color string*)
	visSelectedFlashSegment : ARRAY[0..3] OF USINT := [4(1)]; (*Selected flash segments*)
	visSelectedFlashSegmentOld : ARRAY[0..3] OF USINT := [4(1)]; (*Selected flash segments*)
	visRepetitiveMode : BOOL; (*Enable/Disable repetitive mode*)
	RepetitiveModeTimer : TON; (*Timer for repetitive mode*)
	DisableAutoArchiv : BOOL; (*Enable/Disable automatic archieving for images*)
	InitialSearchSensor : BOOL; (*Flag for first boot*)
	AutoSetupRunning : ARRAY[1..MAX_NUM_CAMS] OF BOOL; (*Flag for auto setup running*)
END_VAR
(*-----------------------------------------------------------------------------------------------------------------------------------------*)
(*Lights variables*)
VAR
	InitialSearchLight : BOOL;
	visLightsTrigger : BOOL;
	visLightsReset : BOOL;
	visLightsEnableCommand : BOOL;
	visLightsFlashColor : STRING[10]; (*Flash color string*)
	visLightsFlashColorOld : STRING[10];
	visEnableLightBarValues : BOOL;
END_VAR
(*-----------------------------------------------------------------------------------------------------------------------------------------*)
(*Code Reader*)
VAR
	visSelectedCodeTypeDetected : ARRAY[1..MAX_NUM_RESULTS] OF STRING[80]; (*HMI helper string*)
	visSelectedCodeType : STRING[80]; (*HMI helper string*)
	visSelectedCodeTypeOld : STRING[80]; (*HMI helper string*)
	visSelectedParameterMode : STRING[80]; (*HMI helper string*)
	visSelectedParameterModeOld : STRING[80]; (*HMI helper string*)
	visCodeTypePresentDropDownValues : ARRAY[0..MAX_NUM_CODETYPES] OF STRING[80];
END_VAR
(*-----------------------------------------------------------------------------------------------------------------------------------------*)
(*Image, crosshair data and constants*)
VAR
	visTableNo : ARRAY[1..MAX_NUM_RESULTS] OF USINT := [1,2,3,4,5,6,7,8,9,10];
	tmpStr1 : STRING[1000];
	i : UINT;
	visCameraStatus : STRING[30];
END_VAR
(*-----------------------------------------------------------------------------------------------------------------------------------------*)
(*Error numbers*)
VAR CONSTANT
	ERR_VA_LIST_NUM : UINT := 30000; (*Number of applications exceeds array size*)
END_VAR
VAR
	visVaListRefresh : BOOL;
END_VAR
```

#### LocalFunctions.fun
```iecst
FUNCTION_BLOCK VaGetList
	VAR_INPUT
		Enable : BOOL;
	END_VAR
	VAR_OUTPUT
		VaApplicationCnt : USINT;
		VaApplicationNames : ARRAY[0..MAX_IDX_VA_LIST] OF STRING[40];
		Status : UINT;
	END_VAR
	VAR
		State : USINT;
	END_VAR
	VAR CONSTANT
		STATE_WAIT : USINT := 0;
		STATE_NEXT_OBJ : USINT := 1;
		STATE_VA_NAME : USINT := 2;
	END_VAR
	VAR
		i : UINT;
		j : UINT;
		PrevIndex : UINT;
		ModuleList : MO_List_typ;
		ModuleStatus : UINT;
		zzEdge00000 : BOOL;
	END_VAR
END_FUNCTION_BLOCK

FUNCTION CrosshairDetailsText : BOOL
	VAR_INPUT
		strTarget : UDINT;
		strText : UDINT;
		fValue : REAL;
	END_VAR
	VAR
		tmpStr : STRING[50];
	END_VAR
END_FUNCTION

FUNCTION String2DataProvider : BOOL
	VAR_INPUT
		SourceString : UDINT;
		TargetString : UDINT;
	END_VAR
END_FUNCTION
```

#### Main.st
```iecst
// --------------------------------------------------------------------------------------------------------------------
// This is a support task for the mappView visualization. The following functions are implemneted
// - Disable mappView functions when camera is not ready, available
// - Transfer parameters after vision setup
// Version 2.x (Check revision history for details)
// --------------------------------------------------------------------------------------------------------------------
PROGRAM _INIT
	// -----------------------------------------------------------------------------------------------------------
	// Map global structure to local reference
	VisionSensor ACCESS ADR(gVisionSensor[gSelectedSensor]);
	Blob ACCESS ADR(tmpBlob);
	CodeReader ACCESS ADR(tmpCodeReader);
	Match ACCESS ADR(tmpMatch);
	MT ACCESS ADR(tmpMT);
	OCR ACCESS ADR(tmpOCR);
	Pixel ACCESS ADR(tmpPixel);

	// Map global structure to local reference
	VisionLight ACCESS ADR(gVisionLight[gSelectedLight]);

	// -----------------------------------------------------------------------------------------------------------
	// Preload code types
	FOR i := 0 TO MAX_NUM_CODETYPES DO
		IF CodeTypes[i] <> '' THEN
			brsstrcat(ADR(visCodeTypePresentDropDownValues[i]), ADR('{"value":"'));
			brsitoa(i, ADR(tmpStr1));
			brsstrcat(ADR(visCodeTypePresentDropDownValues[i]), ADR(tmpStr1));
			brsstrcat(ADR(visCodeTypePresentDropDownValues[i]), ADR('","text":"'));
			brsstrcat(ADR(visCodeTypePresentDropDownValues[i]), ADR(CodeTypes[i]));
			brsstrcat(ADR(visCodeTypePresentDropDownValues[i]), ADR('"}'));
		END_IF
	END_FOR

	// -----------------------------------------------------------------------------------------------------------
	visTableNo;
	InitialSearchSensor := TRUE;
	InitialSearchLight := TRUE;
END_PROGRAM

// -----------------------------------------------------------------------------------------------------------
// Cyclic part
// -----------------------------------------------------------------------------------------------------------
PROGRAM _CYCLIC
	// -----------------------------------------------------------------------------------------------------------
	// Select first available camera after reboot
	// -----------------------------------------------------------------------------------------------------------
	IF InitialSearchSensor THEN
		FOR i := 1 TO MAX_NUM_CAMS DO
			IF gVisionSensor[i].HW.Connected THEN
				gSelectedSensor := i;
				InitialSearchSensor := FALSE;
				EXIT;
			END_IF
		END_FOR
		visVaListRefresh := TRUE;
	END_IF

	// -----------------------------------------------------------------------------------------------------------
	// Map global structure to local reference for mappView
	// -----------------------------------------------------------------------------------------------------------
	// Make sure we dont exceed array limit
	IF(gSelectedSensor > MAX_NUM_CAMS) THEN
		gSelectedSensor := 1;
	END_IF
	IF(gSelectedSensor < 1) THEN
		gSelectedSensor := MAX_NUM_CAMS;
	END_IF
	// -----------------------------------------------------------------------------------------------------------
	// Assign pointers
	VisionSensor ACCESS ADR(gVisionSensor[gSelectedSensor]);
	IF(VisionSensor.CFG.DataStructure <> 0) THEN
		CASE VisionSensor.CFG.VisionFunction OF
			enumBlob:			Blob ACCESS VisionSensor.CFG.DataStructure;
			enumCoderReader:	CodeReader ACCESS VisionSensor.CFG.DataStructure;
			enumMatch:			Match ACCESS VisionSensor.CFG.DataStructure;
			enumMeasurement:	MT ACCESS VisionSensor.CFG.DataStructure;
			enumOCR:			OCR ACCESS VisionSensor.CFG.DataStructure;
			enumPixelCounter:	Pixel ACCESS VisionSensor.CFG.DataStructure;
		END_CASE
	ELSE
		RETURN;
	END_IF

	// -----------------------------------------------------------------------------------------------------------
	// Display camera status
	// -----------------------------------------------------------------------------------------------------------
	visCameraStatus := VisionSensor.DAT.StatusText;

	// -----------------------------------------------------------------------------------------------------------
	// Code Reader - selected/detected types
	// -----------------------------------------------------------------------------------------------------------
	IF VisionSensor.CFG.VisionFunction = enumCoderReader THEN
		IF visSelectedCodeType <> visSelectedCodeTypeOld THEN
			CodeReader.CodeType := UDINT_TO_USINT(brsatoi(ADR(visSelectedCodeType)));
		ELSE
			brsitoa(CodeReader.CodeType, ADR(visSelectedCodeType));
		END_IF
		visSelectedCodeTypeOld := visSelectedCodeType;
		IF visSelectedParameterMode <> visSelectedParameterModeOld THEN
			CodeReader.ParameterMode := UDINT_TO_USINT(brsatoi(ADR(visSelectedParameterMode)));
		ELSE
			brsitoa(CodeReader.ParameterMode, ADR(visSelectedParameterMode));
		END_IF
		visSelectedParameterModeOld := visSelectedParameterMode;
		FOR i := 1 TO MAX_NUM_RESULTS DO
			IF CodeReader.BarcodeType[i] <> 0 THEN
				brsstrcpy(ADR(visSelectedCodeTypeDetected[i]), ADR(CodeTypes[LIMIT(0, CodeReader.BarcodeType[i], MAX_NUM_CODETYPES)]));
			ELSE
				brsstrcpy(ADR(visSelectedCodeTypeDetected[i]), ADR(''));
			END_IF
		END_FOR
	END_IF

	// -----------------------------------------------------------------------------------------------------------
	// Translate flash color and segments from mappView to IO mapping
	// -----------------------------------------------------------------------------------------------------------
	// Hint: Normally copy from recipe (VisionSensor) to visu. Only in case of a change in the visu copy to recipe
	IF visSensorFlashColor <> visSensorFlashColorOld THEN // The flash color was changed in the mappView visualization
		VisionSensor.DAT.FlashColor := UDINT_TO_USINT(brsatoi(ADR(visSensorFlashColor)));
	ELSE
		brsitoa(VisionSensor.DAT.FlashColor, ADR(visSensorFlashColor));
	END_IF
	visSensorFlashColorOld := visSensorFlashColor;
	IF brsmemcmp(ADR(visSelectedFlashSegment), ADR(visSelectedFlashSegmentOld), SIZEOF(visSelectedFlashSegment)) <> 0 THEN // The flash segments was changed in the mappView visualization
		VisionSensor.DAT.FlashSegment := SHL(visSelectedFlashSegment[0], 0) OR SHL(visSelectedFlashSegment[1], 1) OR SHL(visSelectedFlashSegment[2], 2) OR SHL(visSelectedFlashSegment[3], 3);
	ELSE
		visSelectedFlashSegment[0] := VisionSensor.DAT.FlashSegment.0;
		visSelectedFlashSegment[1] := VisionSensor.DAT.FlashSegment.1;
		visSelectedFlashSegment[2] := VisionSensor.DAT.FlashSegment.2;
		visSelectedFlashSegment[3] := VisionSensor.DAT.FlashSegment.3;
	END_IF
	visSelectedFlashSegmentOld := visSelectedFlashSegment;

	// -----------------------------------------------------------------------------------------------------------
	// Disable command buttons when camera is disconnected, not ready, processing an image or vision cockpit is open
	// -----------------------------------------------------------------------------------------------------------
	IF(NOT VisionSensor.HW.Connected OR NOT VisionSensor.HW.Ready OR VisionSensor.DAT.ImageProcessingActive OR VisionSensor.DAT.CockpitIsActive) THEN
		visSensorEnableCommand := FALSE;
	ELSE
		visSensorEnableCommand := TRUE;
	END_IF

	// -----------------------------------------------------------------------------------------------------------
	// Disable setup buttons when camera is disconnected, processing an image or not ready
	// -----------------------------------------------------------------------------------------------------------
	IF(NOT VisionSensor.HW.Connected OR NOT (VisionSensor.HW.Ready OR AutoSetupRunning[gSelectedSensor]) OR VisionSensor.DAT.ImageProcessingActive) THEN
		visEnableSetup := FALSE;
	ELSE
		visEnableSetup := TRUE;
	END_IF

	// -----------------------------------------------------------------------------------------------------------
	// Fire trigger for camera image
	// -----------------------------------------------------------------------------------------------------------
	IF((visImageTrigger OR EDGEPOS(VisionSensor.DAT.Enable)) AND VisionSensor.HW.Ready AND NOT VisionSensor.DAT.ImageProcessingActive) THEN
		// Add default delay and fire trigger
		IF NETTIME_ENABLE THEN
			VisionSensor.DAT.NettimeDelay := NettimeCurrent_us + NETTIME_DEFAULT_DELAY;
		END_IF
		VisionSensor.CMD.ImageTrigger	:= TRUE;
		visImageTrigger					:= FALSE;
		VisionSensor.DAT.Active			:= TRUE;
	END_IF

	// -----------------------------------------------------------------------------------------------------------
	// Auto save image
	// -----------------------------------------------------------------------------------------------------------
	IF EDGENEG(VisionSensor.CMD.ImageTrigger) THEN
		IF visAutoArchiv AND NOT DisableAutoArchiv THEN
			gVisionImage.CMD.SaveImageOnPLC := TRUE;
		END_IF
		IF NOT visRepetitiveMode THEN
			DisableAutoArchiv := FALSE;
		END_IF
	END_IF

	// -----------------------------------------------------------------------------------------------------------
	// Repetitive mode
	// -----------------------------------------------------------------------------------------------------------
	visEnableRepetitive := visSensorEnableCommand OR visRepetitiveMode; // Enable of the repetitive mode button. Don't disable while repetitive mode is active
	IF visRepetitiveMode THEN
		RepetitiveModeTimer.IN := TRUE;
		IF RepetitiveModeTimer.Q THEN
			IF VisionSensor.HW.Ready AND NOT VisionSensor.DAT.ImageProcessingActive THEN
				IF NETTIME_ENABLE THEN
					VisionSensor.DAT.NettimeDelay := NettimeCurrent_us + NETTIME_DEFAULT_DELAY;
				END_IF
				RepetitiveModeTimer.IN := FALSE;
				VisionSensor.CMD.ImageTrigger := TRUE;
			END_IF
		END_IF
		DisableAutoArchiv := TRUE;
		VisionSensor.DAT.Enable := FALSE;
	ELSE
		RepetitiveModeTimer.IN := TRUE;
	END_IF
	RepetitiveModeTimer(PT := T#200ms);

	// -----------------------------------------------------------------------------------------------------------
	// Get list of vision applications and components
	// -----------------------------------------------------------------------------------------------------------
	IF (visVaListRefresh) THEN
		VaGetList_01(Enable := TRUE);
		VisionSensor.FCT.Status := ERR_FUB_BUSY;
		IF VaGetList_01.Status <> ERR_FUB_BUSY THEN
			// Convert vision application list to mappView format
			IF VaGetList_01.Status = ERR_OK THEN
				IF VaGetList_01.VaApplicationCnt > 0 AND VaGetList_01.VaApplicationCnt < MAX_IDX_VA_LIST THEN
					FOR i:=0 TO VaGetList_01.VaApplicationCnt - 1 DO
						String2DataProvider(ADR(VaGetList_01.VaApplicationNames[i]), ADR(visVisionApplicationList[i]));
					END_FOR
				END_IF
				VisionSensor.FCT.Status := ERR_OK;
			ELSE // Error
				brsmemset(ADR(visVisionApplicationList), 0, SIZEOF(visVisionApplicationList));
				VisionSensor.FCT.Status := VaGetList_01.Status;
			END_IF
			// Reset function block
			VaGetList_01(Enable := FALSE);
			visVaListRefresh := FALSE;
		END_IF
	END_IF

	// -----------------------------------------------------------------------------------------------------------
	// Select first available light after reboot
	// -----------------------------------------------------------------------------------------------------------
	IF InitialSearchLight THEN
		FOR i := 1 TO MAX_NUM_LIGHTS DO
			IF gVisionLight[i].HW.Connected THEN
				gSelectedLight := i;
				InitialSearchLight := FALSE;
				EXIT;
			END_IF
		END_FOR
	END_IF
	// -----------------------------------------------------------------------------------------------------------
	// Map global structure to local reference
	// -----------------------------------------------------------------------------------------------------------
	// Make sure we dont exceed array limit
	IF(gSelectedLight > MAX_NUM_LIGHTS) THEN
		gSelectedLight := 1;
	END_IF
	IF(gSelectedLight < 1) THEN
		gSelectedLight := MAX_NUM_LIGHTS;
	END_IF
	VisionLight ACCESS ADR(gVisionLight[gSelectedLight]);

	// -----------------------------------------------------------------------------------------------------------
	// Translate flash color from mappView to IO mapping
	// -----------------------------------------------------------------------------------------------------------
	// Hint: Normally copy from recipe (VisionLight) to visu. Only in case of a change in the visu copy to recipe
	IF visLightsFlashColor <> visLightsFlashColorOld THEN // The flash color was changed in the mappView visualization
		VisionLight.DAT.FlashColor := UDINT_TO_USINT(brsatoi(ADR(visLightsFlashColor)));
	ELSE
		brsitoa(VisionLight.DAT.FlashColor, ADR(visLightsFlashColor));
	END_IF
	visLightsFlashColorOld := visLightsFlashColor;

	// -----------------------------------------------------------------------------------------------------------
	// Reset Light trigger manually
	// -----------------------------------------------------------------------------------------------------------
	IF (visLightsReset) THEN
		VisionLight.CMD.FlashTrigger := FALSE;
		visLightsReset := FALSE;
	END_IF

	// -----------------------------------------------------------------------------------------------------------
	// Fire trigger for lights
	// -----------------------------------------------------------------------------------------------------------
	IF(visLightsTrigger AND VisionLight.HW.Ready) THEN
		// Add default delay and fire trigger
		IF NETTIME_ENABLE THEN
			VisionLight.DAT.NettimeDelay := NettimeCurrent_us + NETTIME_DEFAULT_DELAY;
		END_IF
		VisionLight.CMD.FlashTrigger := TRUE;
		visLightsTrigger := FALSE;
	END_IF

	// -----------------------------------------------------------------------------------------------------------
	// Disable command button when light is disconnected or not ready
	// -----------------------------------------------------------------------------------------------------------
	IF(NOT VisionLight.HW.Connected OR NOT VisionLight.HW.Ready) THEN
		visLightsEnableCommand := FALSE;
	ELSE
		visLightsEnableCommand := TRUE;
	END_IF

	// -----------------------------------------------------------------------------------------------------------
	// Enable fields for different light types
	// -----------------------------------------------------------------------------------------------------------
	visEnableLightBarValues := VisionLight.CFG.LightType = enumLightbar;
END_PROGRAM
```

### Program Logical/old/YourTask

#### Variables.var
```iecst
VAR
	visNewRecipe : BOOL; (*New camera settings recipe*)
	visSaveRecipe : BOOL; (*Save camera settings*)
	cmdLoadRecipeAfterBoot : BOOL;
	i : INT;
END_VAR
```
